  MoveL 8129 to (238.13, 41.99, 116.27) mm, rotated rx 180 ry 0 rz 180 deg; joints [-18.333, 8.057, 71.55, 61.436, 20.986, -59.754]
  Call Extruder(204.42198)
  MoveL 8130 to (238.31, 42.3, 116.27) mm, rotated rx 180 ry 0 rz 180 deg; joints [-18.36, 8.102, 71.5, 61.459, 21.011, -59.774]
  MoveL 8131 to (238.31, 42.3, 116.27) mm, rotated rx 180 ry 0 rz 180 deg; joints [-18.36, 8.102, 71.5, 61.459, 21.011, -59.774]
  Call Extruder(204.62931)
  MoveL 8132 to (238.49, 42.6, 116.27) mm, rotated rx 180 ry 0 rz 180 deg; joints [-18.386, 8.146, 71.449, 61.482, 21.037, -59.794]
  MoveL 8133 to (238.49, 42.6, 116.27) mm, rotated rx 180 ry 0 rz 180 deg; joints [-18.386, 8.146, 71.449, 61.482, 21.037, -59.794]
  Call Extruder(204.83587)
  MoveL 8134 to (238.66, 42.91, 116.27) mm, rotated rx 180 ry 0 rz 180 deg; joints [-18.412, 8.19, 71.399, 61.505, 21.062, -59.813]
  MoveL 8135 to (238.66, 42.91, 116.27) mm, rotated rx 180 ry 0 rz 180 deg; joints [-18.412, 8.19, 71.399, 61.505, 21.062, -59.813]
  Call Extruder(205.04165)
  MoveL 8136 to (238.84, 43.21, 116.27) mm, rotated rx 180 ry 0 rz -180 deg; joints [-18.438, 8.235, 71.349, 61.528, 21.088, -59.833]
  MoveL 8137 to (238.84, 43.21, 116.27) mm, rotated rx 180 ry 0 rz -180 deg; joints [-18.438, 8.235, 71.349, 61.528, 21.088, -59.833]
  Call Extruder(205.19996)
  MoveL 8138 to (238.94, 43.46, 116.27) mm, rotated rx 180 ry 0 rz 180 deg; joints [-18.461, 8.265, 71.314, 61.55, 21.11, -59.852]
  MoveL 8139 to (238.94, 43.46, 116.27) mm, rotated rx 180 ry 0 rz 180 deg; joints [-18.461, 8.265, 71.314, 61.55, 21.11, -59.852]
  Call Extruder(205.35767)
  MoveL 8140 to (239.05, 43.71, 116.27) mm, rotated rx 180 ry 0 rz 180 deg; joints [-18.484, 8.296, 71.279, 61.573, 21.131, -59.872]
  MoveL 8141 to (239.05, 43.71, 116.27) mm, rotated rx 180 ry 0 rz 180 deg; joints [-18.484, 8.296, 71.279, 61.573, 21.131, -59.872]
  Call Extruder(205.52776)
  MoveL 8142 to (239.16, 43.98, 116.27) mm, rotated rx 180 ry 0 rz 180 deg; joints [-18.509, 8.328, 71.242, 61.597, 21.155, -59.893]
  MoveL 8143 to (239.16, 43.98, 116.27) mm, rotated rx 180 ry 0 rz 180 deg; joints [-18.509, 8.328, 71.242, 61.597, 21.155, -59.893]
  Call Extruder(205.71010)
  MoveL 8144 to (239.29, 44.27, 116.27) mm, rotated rx 180 ry 0 rz -180 deg; joints [-18.535, 8.363, 71.202, 61.623, 21.18, -59.916]
  MoveL 8145 to (239.29, 44.27, 116.27) mm, rotated rx 180 ry 0 rz -180 deg; joints [-18.535, 8.363, 71.202, 61.623, 21.18, -59.916]
  Call Extruder(205.89168)
  MoveL 8146 to (239.41, 44.56, 116.27) mm, rotated rx 180 ry 0 rz 180 deg; joints [-18.562, 8.399, 71.162, 61.649, 21.206, -59.938]
  MoveL 8147 to (239.41, 44.56, 116.27) mm, rotated rx 180 ry 0 rz 180 deg; joints [-18.562, 8.399, 71.162, 61.649, 21.206, -59.938]
  Call Extruder(206.00513)
  MoveL 8148 to (239.47, 44.75, 116.27) mm, rotated rx -180 ry 0 rz 180 deg; joints [-18.58, 8.418, 71.139, 61.667, 21.223, -59.954]
  MoveL 8149 to (239.47, 44.75, 116.27) mm, rotated rx -180 ry 0 rz 180 deg; joints [-18.58, 8.418, 71.139, 61.667, 21.223, -59.954]
  Call Extruder(206.11815)
  MoveL 8150 to (239.53, 44.94, 116.27) mm, rotated rx 180 ry 0 rz 180 deg; joints [-18.598, 8.438, 71.116, 61.686, 21.239, -59.971]
  MoveL 8151 to (239.53, 44.94, 116.27) mm, rotated rx 180 ry 0 rz 180 deg; joints [-18.598, 8.438, 71.116, 61.686, 21.239, -59.971]
  Call Extruder(206.23072)
  MoveL 8152 to (239.59, 45.13, 116.27) mm, rotated rx 180 ry 0 rz -180 deg; joints [-18.616, 8.459, 71.093, 61.704, 21.256, -59.987]
  MoveL 8153 to (239.59, 45.13, 116.27) mm, rotated rx 180 ry 0 rz -180 deg; joints [-18.616, 8.459, 71.093, 61.704, 21.256, -59.987]
  Call Extruder(206.34284)
  MoveL 8154 to (239.65, 45.32, 116.27) mm, rotated rx -180 ry 0 rz 180 deg; joints [-18.634, 8.479, 71.071, 61.722, 21.273, -60.003]
  MoveL 8155 to (239.65, 45.32, 116.27) mm, rotated rx -180 ry 0 rz 180 deg; joints [-18.634, 8.479, 71.071, 61.722, 21.273, -60.003]
  Call Extruder(206.45452)
  MoveL 8156 to (239.71, 45.51, 116.27) mm, rotated rx -180 ry 0 rz 180 deg; joints [-18.651, 8.499, 71.048, 61.74, 21.29, -60.019]
  MoveL 8157 to (239.71, 45.51, 116.27) mm, rotated rx -180 ry 0 rz 180 deg; joints [-18.651, 8.499, 71.048, 61.74, 21.29, -60.019]
  Call Extruder(206.58559)
  MoveL 8158 to (239.78, 45.73, 116.27) mm, rotated rx 180 ry 0 rz 180 deg; joints [-18.673, 8.522, 71.022, 61.762, 21.31, -60.038]
  MoveL 8159 to (239.78, 45.73, 116.27) mm, rotated rx 180 ry 0 rz 180 deg; joints [-18.673, 8.522, 71.022, 61.762, 21.31, -60.038]
  Call Extruder(206.71610)
  MoveL 8160 to (239.85, 45.95, 116.27) mm, rotated rx 180 ry 0 rz -180 deg; joints [-18.694, 8.545, 70.995, 61.784, 21.33, -60.058]
  MoveL 8161 to (239.85, 45.95, 116.27) mm, rotated rx 180 ry 0 rz -180 deg; joints [-18.694, 8.545, 70.995, 61.784, 21.33, -60.058]
  Call Extruder(206.84604)
  MoveL 8162 to (239.92, 46.18, 116.27) mm, rotated rx 180 ry 0 rz -180 deg; joints [-18.715, 8.568, 70.969, 61.806, 21.35, -60.077]
  MoveL 8163 to (239.92, 46.18, 116.27) mm, rotated rx 180 ry 0 rz -180 deg; joints [-18.715, 8.568, 70.969, 61.806, 21.35, -60.077]
  Call Extruder(206.97542)
  MoveL 8164 to (239.98, 46.4, 116.27) mm, rotated rx -180 ry 0 rz -180 deg; joints [-18.737, 8.591, 70.943, 61.828, 21.37, -60.096]
  MoveL 8165 to (239.98, 46.4, 116.27) mm, rotated rx -180 ry 0 rz -180 deg; joints [-18.737, 8.591, 70.943, 61.828, 21.37, -60.096]
  Call Extruder(207.09738)
  MoveL 8166 to (240.04, 46.61, 116.27) mm, rotated rx -180 ry 0 rz 180 deg; joints [-18.757, 8.611, 70.919, 61.849, 21.389, -60.115]
  MoveL 8167 to (240.04, 46.61, 116.27) mm, rotated rx -180 ry 0 rz 180 deg; joints [-18.757, 8.611, 70.919, 61.849, 21.389, -60.115]
  Call Extruder(207.21220)
  MoveL 8168 to (240.08, 46.82, 116.27) mm, rotated rx 180 ry 0 rz 180 deg; joints [-18.777, 8.63, 70.898, 61.871, 21.408, -60.135]
  MoveL 8169 to (240.08, 46.82, 116.27) mm, rotated rx 180 ry 0 rz 180 deg; joints [-18.777, 8.63, 70.898, 61.871, 21.408, -60.135]
  Call Extruder(207.32658)
  MoveL 8170 to (240.13, 47.02, 116.27) mm, rotated rx -180 ry 0 rz 180 deg; joints [-18.797, 8.648, 70.877, 61.892, 21.426, -60.154]
  MoveL 8171 to (240.13, 47.02, 116.27) mm, rotated rx -180 ry 0 rz 180 deg; joints [-18.797, 8.648, 70.877, 61.892, 21.426, -60.154]
  Call Extruder(207.44050)
  MoveL 8172 to (240.17, 47.23, 116.27) mm, rotated rx 180 ry 0 rz 180 deg; joints [-18.817, 8.666, 70.856, 61.913, 21.445, -60.173]
  MoveL 8173 to (240.17, 47.23, 116.27) mm, rotated rx 180 ry 0 rz 180 deg; joints [-18.817, 8.666, 70.856, 61.913, 21.445, -60.173]
  Call Extruder(207.55397)
  MoveL 8174 to (240.22, 47.43, 116.27) mm, rotated rx 180 ry 0 rz 180 deg; joints [-18.837, 8.685, 70.835, 61.935, 21.464, -60.192]
  MoveL 8175 to (240.22, 47.43, 116.27) mm, rotated rx 180 ry 0 rz 180 deg; joints [-18.837, 8.685, 70.835, 61.935, 21.464, -60.192]
  Call Extruder(207.69125)
  MoveL 8176 to (240.27, 47.68, 116.27) mm, rotated rx 180 ry 0 rz -180 deg; joints [-18.862, 8.706, 70.81, 61.961, 21.486, -60.215]
  MoveL 8177 to (240.27, 47.68, 116.27) mm, rotated rx 180 ry 0 rz -180 deg; joints [-18.862, 8.706, 70.81, 61.961, 21.486, -60.215]
  Call Extruder(207.82792)
  MoveL 8178 to (240.32, 47.93, 116.27) mm, rotated rx 180 ry 0 rz 180 deg; joints [-18.887, 8.728, 70.786, 61.987, 21.509, -60.239]
  MoveL 8179 to (240.32, 47.93, 116.27) mm, rotated rx 180 ry 0 rz 180 deg; joints [-18.887, 8.728, 70.786, 61.987, 21.509, -60.239]
  Call Extruder(207.96399)
  MoveL 8180 to (240.37, 48.18, 116.27) mm, rotated rx 180 ry 0 rz 180 deg; joints [-18.911, 8.75, 70.761, 62.014, 21.532, -60.262]
  MoveL 8181 to (240.37, 48.18, 116.27) mm, rotated rx 180 ry 0 rz 180 deg; joints [-18.911, 8.75, 70.761, 62.014, 21.532, -60.262]
  Call Extruder(208.09944)
  MoveL 8182 to (240.42, 48.43, 116.27) mm, rotated rx 180 ry 0 rz 180 deg; joints [-18.936, 8.771, 70.736, 62.04, 21.555, -60.285]
  MoveL 8183 to (240.42, 48.43, 116.27) mm, rotated rx 180 ry 0 rz 180 deg; joints [-18.936, 8.771, 70.736, 62.04, 21.555, -60.285]
  Call Extruder(208.23428)
  MoveL 8184 to (240.47, 48.68, 116.27) mm, rotated rx 180 ry 0 rz -180 deg; joints [-18.96, 8.793, 70.711, 62.066, 21.578, -60.308]
  MoveL 8185 to (240.47, 48.68, 116.27) mm, rotated rx 180 ry 0 rz -180 deg; joints [-18.96, 8.793, 70.711, 62.066, 21.578, -60.308]
  Call Extruder(208.36851)
  MoveL 8186 to (240.52, 48.92, 116.27) mm, rotated rx 180 ry 0 rz 180 deg; joints [-18.985, 8.815, 70.686, 62.092, 21.6, -60.331]
  MoveL 8187 to (240.52, 48.92, 116.27) mm, rotated rx 180 ry 0 rz 180 deg; joints [-18.985, 8.815, 70.686, 62.092, 21.6, -60.331]
  Call Extruder(208.50213)
  MoveL 8188 to (240.57, 49.17, 116.27) mm, rotated rx 180 ry 0 rz 180 deg; joints [-19.009, 8.837, 70.661, 62.117, 21.623, -60.354]
  MoveL 8189 to (240.57, 49.17, 116.27) mm, rotated rx 180 ry 0 rz 180 deg; joints [-19.009, 8.837, 70.661, 62.117, 21.623, -60.354]
  Call Extruder(208.66424)
  MoveL 8190 to (240.61, 49.48, 116.27) mm, rotated rx -180 ry 0 rz 180 deg; joints [-19.04, 8.861, 70.633, 62.15, 21.651, -60.384]
  MoveL 8191 to (240.61, 49.48, 116.27) mm, rotated rx -180 ry 0 rz 180 deg; joints [-19.04, 8.861, 70.633, 62.15, 21.651, -60.384]
  Call Extruder(208.82562)
  MoveL 8192 to (240.66, 49.79, 116.27) mm, rotated rx 180 ry 0 rz 180 deg; joints [-19.07, 8.886, 70.604, 62.183, 21.68, -60.413]
  MoveL 8193 to (240.66, 49.79, 116.27) mm, rotated rx 180 ry 0 rz 180 deg; joints [-19.07, 8.886, 70.604, 62.183, 21.68, -60.413]
  Call Extruder(208.98628)
  MoveL 8194 to (240.71, 50.09, 116.27) mm, rotated rx 180 ry 0 rz 180 deg; joints [-19.101, 8.911, 70.576, 62.215, 21.708, -60.442]
  MoveL 8195 to (240.71, 50.09, 116.27) mm, rotated rx 180 ry 0 rz 180 deg; joints [-19.101, 8.911, 70.576, 62.215, 21.708, -60.442]
  Call Extruder(209.14620)
  MoveL 8196 to (240.76, 50.4, 116.27) mm, rotated rx 180 ry 0 rz 180 deg; joints [-19.131, 8.936, 70.547, 62.248, 21.736, -60.471]
  MoveL 8197 to (240.76, 50.4, 116.27) mm, rotated rx 180 ry 0 rz 180 deg; joints [-19.131, 8.936, 70.547, 62.248, 21.736, -60.471]
  Call Extruder(209.30540)
  MoveL 8198 to (240.81, 50.7, 116.27) mm, rotated rx 180 ry 0 rz -180 deg; joints [-19.162, 8.961, 70.519, 62.28, 21.764, -60.499]
  MoveL 8199 to (240.81, 50.7, 116.27) mm, rotated rx 180 ry 0 rz -180 deg; joints [-19.162, 8.961, 70.519, 62.28, 21.764, -60.499]
  Call Extruder(209.46387)
  MoveL 8200 to (240.86, 51.01, 116.27) mm, rotated rx 180 ry 0 rz 180 deg; joints [-19.192, 8.986, 70.49, 62.312, 21.793, -60.528]
  MoveL 8201 to (240.86, 51.01, 116.27) mm, rotated rx 180 ry 0 rz 180 deg; joints [-19.192, 8.986, 70.49, 62.312, 21.793, -60.528]
  Call Extruder(209.66274)
  MoveL 8202 to (240.9, 51.4, 116.27) mm, rotated rx 180 ry 0 rz 180 deg; joints [-19.231, 9.015, 70.457, 62.354, 21.829, -60.566]
  MoveL 8203 to (240.9, 51.4, 116.27) mm, rotated rx 180 ry 0 rz 180 deg; joints [-19.231, 9.015, 70.457, 62.354, 21.829, -60.566]
  Call Extruder(209.86075)
  MoveL 8204 to (240.95, 51.78, 116.27) mm, rotated rx 180 ry 0 rz 180 deg; joints [-19.27, 9.044, 70.423, 62.396, 21.865, -60.603]
  MoveL 8205 to (240.95, 51.78, 116.27) mm, rotated rx 180 ry 0 rz 180 deg; joints [-19.27, 9.044, 70.423, 62.396, 21.865, -60.603]
  Call Extruder(210.05789)
  MoveL 8206 to (240.99, 52.17, 116.27) mm, rotated rx 180 ry 0 rz -180 deg; joints [-19.309, 9.073, 70.389, 62.438, 21.901, -60.64]
  MoveL 8207 to (240.99, 52.17, 116.27) mm, rotated rx 180 ry 0 rz -180 deg; joints [-19.309, 9.073, 70.389, 62.438, 21.901, -60.64]
  Call Extruder(210.25416)
  MoveL 8208 to (241.04, 52.56, 116.27) mm, rotated rx 180 ry 0 rz 180 deg; joints [-19.348, 9.102, 70.356, 62.48, 21.937, -60.678]
  MoveL 8209 to (241.04, 52.56, 116.27) mm, rotated rx 180 ry 0 rz 180 deg; joints [-19.348, 9.102, 70.356, 62.48, 21.937, -60.678]
  Call Extruder(210.49987)
  MoveL 8210 to (241.09, 53.05, 116.27) mm, rotated rx 180 ry 0 rz 180 deg; joints [-19.398, 9.137, 70.315, 62.533, 21.983, -60.725]
  MoveL 8211 to (241.09, 53.05, 116.27) mm, rotated rx 180 ry 0 rz 180 deg; joints [-19.398, 9.137, 70.315, 62.533, 21.983, -60.725]
  Call Extruder(210.79465)
  MoveL 8212 to (241.13, 53.64, 116.27) mm, rotated rx 180 ry 0 rz 180 deg; joints [-19.458, 9.178, 70.268, 62.598, 22.038, -60.783]
  MoveL 8213 to (241.13, 53.64, 116.27) mm, rotated rx 180 ry 0 rz 180 deg; joints [-19.458, 9.178, 70.268, 62.598, 22.038, -60.783]
  Call Extruder(211.08809)
  MoveL 8214 to (241.18, 54.23, 116.27) mm, rotated rx 180 ry 0 rz 180 deg; joints [-19.518, 9.219, 70.221, 62.662, 22.093, -60.84]
  MoveL 8215 to (241.18, 54.23, 116.27) mm, rotated rx 180 ry 0 rz 180 deg; joints [-19.518, 9.219, 70.221, 62.662, 22.093, -60.84]
  Call Extruder(211.52144)
  MoveL 8216 to (241.22, 55.1, 116.27) mm, rotated rx 180 ry 0 rz 180 deg; joints [-19.608, 9.277, 70.154, 62.759, 22.176, -60.927]
  MoveL 8217 to (241.22, 55.1, 116.27) mm, rotated rx 180 ry 0 rz 180 deg; joints [-19.608, 9.277, 70.154, 62.759, 22.176, -60.927]
  Call Extruder(212.09360)
  MoveL 8218 to (241.27, 56.26, 116.27) mm, rotated rx 180 ry 0 rz 180 deg; joints [-19.728, 9.351, 70.069, 62.888, 22.286, -61.043]
  MoveL 8219 to (241.27, 56.26, 116.27) mm, rotated rx 180 ry 0 rz 180 deg; joints [-19.728, 9.351, 70.069, 62.888, 22.286, -61.043]
  Call Extruder(212.52130)
  MoveL 8220 to (241.29, 57.14, 116.27) mm, rotated rx 180 ry 0 rz 180 deg; joints [-19.819, 9.405, 70.007, 62.985, 22.369, -61.13]
  Call Extruder(254.51494)
  MoveL 8221 to (241.29, 142.86, 116.27) mm, rotated rx 180 ry 0 rz 180 deg; joints [-28.232, 15.645, 62.466, 69.008, 30.442, -66.009]
  MoveL 8222 to (241.29, 142.86, 116.27) mm, rotated rx 180 ry 0 rz 180 deg; joints [-28.232, 15.645, 62.466, 69.008, 30.442, -66.009]
  Call Extruder(255.23038)
  MoveL 8223 to (241.25, 144.32, 116.27) mm, rotated rx 180 ry 0 rz 180 deg; joints [-28.367, 15.768, 62.311, 69.066, 30.577, -66.043]
  MoveL 8224 to (241.25, 144.32, 116.27) mm, rotated rx 180 ry 0 rz 180 deg; joints [-28.367, 15.768, 62.311, 69.066, 30.577, -66.043]
  Call Extruder(255.80512)
  MoveL 8225 to (241.2, 145.48, 116.27) mm, rotated rx 180 ry 0 rz 180 deg; joints [-28.475, 15.864, 62.19, 69.112, 30.685, -66.071]
  MoveL 8226 to (241.2, 145.48, 116.27) mm, rotated rx 180 ry 0 rz 180 deg; joints [-28.475, 15.864, 62.19, 69.112, 30.685, -66.071]
  Call Extruder(256.09856)
  MoveL 8227 to (241.15, 146.07, 116.27) mm, rotated rx 180 ry 0 rz 180 deg; joints [-28.531, 15.909, 62.133, 69.138, 30.741, -66.087]
  MoveL 8228 to (241.15, 146.07, 116.27) mm, rotated rx 180 ry 0 rz 180 deg; joints [-28.531, 15.909, 62.133, 69.138, 30.741, -66.087]
  Call Extruder(256.39333)
  MoveL 8229 to (241.11, 146.66, 116.27) mm, rotated rx 180 ry 0 rz 180 deg; joints [-28.587, 15.954, 62.076, 69.163, 30.796, -66.103]
  MoveL 8230 to (241.11, 146.66, 116.27) mm, rotated rx 180 ry 0 rz 180 deg; joints [-28.587, 15.954, 62.076, 69.163, 30.796, -66.103]
  Call Extruder(256.68944)
  MoveL 8231 to (241.06, 147.25, 116.27) mm, rotated rx 180 ry 0 rz 180 deg; joints [-28.643, 15.999, 62.018, 69.189, 30.852, -66.119]
  MoveL 8232 to (241.06, 147.25, 116.27) mm, rotated rx 180 ry 0 rz 180 deg; joints [-28.643, 15.999, 62.018, 69.189, 30.852, -66.119]
  Call Extruder(256.88571)
  MoveL 8233 to (241.02, 147.63, 116.27) mm, rotated rx -180 ry 0 rz 180 deg; joints [-28.681, 16.027, 61.984, 69.207, 30.888, -66.131]
  MoveL 8234 to (241.02, 147.63, 116.27) mm, rotated rx -180 ry 0 rz 180 deg; joints [-28.681, 16.027, 61.984, 69.207, 30.888, -66.131]
  Call Extruder(257.08285)
  MoveL 8235 to (240.97, 148.02, 116.27) mm, rotated rx -180 ry 0 rz 180 deg; joints [-28.718, 16.054, 61.949, 69.225, 30.925, -66.143]
  MoveL 8236 to (240.97, 148.02, 116.27) mm, rotated rx -180 ry 0 rz 180 deg; joints [-28.718, 16.054, 61.949, 69.225, 30.925, -66.143]
  Call Extruder(257.28085)
  MoveL 8237 to (240.92, 148.41, 116.27) mm, rotated rx -180 ry 0 rz 180 deg; joints [-28.756, 16.082, 61.914, 69.243, 30.962, -66.155]
  MoveL 8238 to (240.92, 148.41, 116.27) mm, rotated rx -180 ry 0 rz 180 deg; joints [-28.756, 16.082, 61.914, 69.243, 30.962, -66.155]
  Call Extruder(257.47973)
  MoveL 8239 to (240.88, 148.8, 116.27) mm, rotated rx 180 ry 0 rz 180 deg; joints [-28.793, 16.109, 61.879, 69.261, 30.999, -66.167]
  MoveL 8240 to (240.88, 148.8, 116.27) mm, rotated rx 180 ry 0 rz 180 deg; joints [-28.793, 16.109, 61.879, 69.261, 30.999, -66.167]
  Call Extruder(257.65881)
  MoveL 8241 to (240.83, 149.14, 116.27) mm, rotated rx -180 ry 0 rz 180 deg; joints [-28.827, 16.133, 61.849, 69.277, 31.032, -66.178]
  MoveL 8242 to (240.83, 149.14, 116.27) mm, rotated rx -180 ry 0 rz 180 deg; joints [-28.827, 16.133, 61.849, 69.277, 31.032, -66.178]
  Call Extruder(257.81801)
  MoveL 8243 to (240.78, 149.45, 116.27) mm, rotated rx 180 ry 0 rz 180 deg; joints [-28.857, 16.153, 61.824, 69.293, 31.062, -66.189]
  MoveL 8244 to (240.78, 149.45, 116.27) mm, rotated rx 180 ry 0 rz 180 deg; joints [-28.857, 16.153, 61.824, 69.293, 31.062, -66.189]
  Call Extruder(257.97794)
  MoveL 8245 to (240.74, 149.76, 116.27) mm, rotated rx 180 ry 0 rz 180 deg; joints [-28.887, 16.173, 61.799, 69.308, 31.091, -66.199]
  MoveL 8246 to (240.74, 149.76, 116.27) mm, rotated rx 180 ry 0 rz 180 deg; joints [-28.887, 16.173, 61.799, 69.308, 31.091, -66.199]
  Call Extruder(258.13859)
  MoveL 8247 to (240.69, 150.06, 116.27) mm, rotated rx 180 ry 0 rz 180 deg; joints [-28.917, 16.192, 61.774, 69.323, 31.12, -66.21]
  MoveL 8248 to (240.69, 150.06, 116.27) mm, rotated rx 180 ry 0 rz 180 deg; joints [-28.917, 16.192, 61.774, 69.323, 31.12, -66.21]
  Call Extruder(258.29997)
  MoveL 8249 to (240.64, 150.37, 116.27) mm, rotated rx 180 ry 0 rz 180 deg; joints [-28.947, 16.212, 61.749, 69.338, 31.15, -66.22]
  MoveL 8250 to (240.64, 150.37, 116.27) mm, rotated rx 180 ry 0 rz 180 deg; joints [-28.947, 16.212, 61.749, 69.338, 31.15, -66.22]
  Call Extruder(258.46208)
  MoveL 8251 to (240.59, 150.67, 116.27) mm, rotated rx -180 ry 0 rz 180 deg; joints [-28.978, 16.232, 61.723, 69.353, 31.179, -66.23]
  MoveL 8252 to (240.59, 150.67, 116.27) mm, rotated rx -180 ry 0 rz 180 deg; joints [-28.978, 16.232, 61.723, 69.353, 31.179, -66.23]
  Call Extruder(258.61028)
  MoveL 8253 to (240.54, 150.95, 116.27) mm, rotated rx -180 ry 0 rz 180 deg; joints [-29.005, 16.249, 61.701, 69.368, 31.206, -66.24]
  MoveL 8254 to (240.54, 150.95, 116.27) mm, rotated rx -180 ry 0 rz 180 deg; joints [-29.005, 16.249, 61.701, 69.368, 31.206, -66.24]
  Call Extruder(258.74452)
  MoveL 8255 to (240.49, 151.2, 116.27) mm, rotated rx 180 ry 0 rz 180 deg; joints [-29.03, 16.264, 61.683, 69.381, 31.23, -66.25]
  MoveL 8256 to (240.49, 151.2, 116.27) mm, rotated rx 180 ry 0 rz 180 deg; joints [-29.03, 16.264, 61.683, 69.381, 31.23, -66.25]
  Call Extruder(258.87936)
  MoveL 8257 to (240.44, 151.45, 116.27) mm, rotated rx 180 ry 0 rz 180 deg; joints [-29.055, 16.279, 61.664, 69.394, 31.255, -66.259]
  MoveL 8258 to (240.44, 151.45, 116.27) mm, rotated rx 180 ry 0 rz 180 deg; joints [-29.055, 16.279, 61.664, 69.394, 31.255, -66.259]
  Call Extruder(259.01481)
  MoveL 8259 to (240.39, 151.7, 116.27) mm, rotated rx -180 ry 0 rz 180 deg; joints [-29.08, 16.293, 61.646, 69.407, 31.279, -66.268]
  MoveL 8260 to (240.39, 151.7, 116.27) mm, rotated rx -180 ry 0 rz 180 deg; joints [-29.08, 16.293, 61.646, 69.407, 31.279, -66.268]
  Call Extruder(259.15087)
  MoveL 8261 to (240.34, 151.95, 116.27) mm, rotated rx 180 ry 0 rz 180 deg; joints [-29.105, 16.308, 61.627, 69.421, 31.303, -66.278]
  MoveL 8262 to (240.34, 151.95, 116.27) mm, rotated rx 180 ry 0 rz 180 deg; joints [-29.105, 16.308, 61.627, 69.421, 31.303, -66.278]
  Call Extruder(259.28754)
  MoveL 8263 to (240.29, 152.2, 116.27) mm, rotated rx 180 ry 0 rz 180 deg; joints [-29.13, 16.323, 61.608, 69.434, 31.327, -66.287]
  MoveL 8264 to (240.29, 152.2, 116.27) mm, rotated rx 180 ry 0 rz 180 deg; joints [-29.13, 16.323, 61.608, 69.434, 31.327, -66.287]
  Call Extruder(259.42483)
  MoveL 8265 to (240.24, 152.44, 116.27) mm, rotated rx 180 ry 0 rz 180 deg; joints [-29.155, 16.338, 61.589, 69.447, 31.352, -66.296]
  MoveL 8266 to (240.24, 152.44, 116.27) mm, rotated rx 180 ry 0 rz 180 deg; joints [-29.155, 16.338, 61.589, 69.447, 31.352, -66.296]
  Call Extruder(259.55049)
  MoveL 8267 to (240.2, 152.67, 116.27) mm, rotated rx -180 ry 0 rz 180 deg; joints [-29.178, 16.351, 61.573, 69.459, 31.374, -66.305]
  MoveL 8268 to (240.2, 152.67, 116.27) mm, rotated rx -180 ry 0 rz 180 deg; joints [-29.178, 16.351, 61.573, 69.459, 31.374, -66.305]
  Call Extruder(259.66441)
  MoveL 8269 to (240.15, 152.88, 116.27) mm, rotated rx 180 ry 0 rz -180 deg; joints [-29.198, 16.362, 61.558, 69.47, 31.394, -66.313]
  MoveL 8270 to (240.15, 152.88, 116.27) mm, rotated rx 180 ry 0 rz -180 deg; joints [-29.198, 16.362, 61.558, 69.47, 31.394, -66.313]
  Call Extruder(259.77879)
  MoveL 8271 to (240.11, 153.08, 116.27) mm, rotated rx 180 ry 0 rz 180 deg; joints [-29.219, 16.374, 61.543, 69.481, 31.414, -66.321]
  MoveL 8272 to (240.11, 153.08, 116.27) mm, rotated rx 180 ry 0 rz 180 deg; joints [-29.219, 16.374, 61.543, 69.481, 31.414, -66.321]
  Call Extruder(259.89362)
  MoveL 8273 to (240.06, 153.28, 116.27) mm, rotated rx 180 ry 0 rz 180 deg; joints [-29.24, 16.385, 61.529, 69.492, 31.434, -66.329]
  MoveL 8274 to (240.06, 153.28, 116.27) mm, rotated rx 180 ry 0 rz 180 deg; joints [-29.24, 16.385, 61.529, 69.492, 31.434, -66.329]
  Call Extruder(260.00890)
  MoveL 8275 to (240.02, 153.49, 116.27) mm, rotated rx -180 ry 0 rz 180 deg; joints [-29.26, 16.396, 61.514, 69.503, 31.454, -66.337]
  MoveL 8276 to (240.02, 153.49, 116.27) mm, rotated rx -180 ry 0 rz 180 deg; joints [-29.26, 16.396, 61.514, 69.503, 31.454, -66.337]
  Call Extruder(260.13828)
  MoveL 8277 to (239.95, 153.71, 116.27) mm, rotated rx -180 ry 0 rz 180 deg; joints [-29.284, 16.406, 61.502, 69.518, 31.476, -66.347]
  MoveL 8278 to (239.95, 153.71, 116.27) mm, rotated rx -180 ry 0 rz 180 deg; joints [-29.284, 16.406, 61.502, 69.518, 31.476, -66.347]
  Call Extruder(260.26822)
  MoveL 8279 to (239.88, 153.94, 116.27) mm, rotated rx -180 ry 0 rz 180 deg; joints [-29.307, 16.416, 61.49, 69.532, 31.499, -66.358]
  MoveL 8280 to (239.88, 153.94, 116.27) mm, rotated rx -180 ry 0 rz 180 deg; joints [-29.307, 16.416, 61.49, 69.532, 31.499, -66.358]
  Call Extruder(260.39873)
  MoveL 8281 to (239.82, 154.16, 116.27) mm, rotated rx 180 ry 0 rz 180 deg; joints [-29.331, 16.425, 61.478, 69.546, 31.521, -66.369]
  MoveL 8282 to (239.82, 154.16, 116.27) mm, rotated rx 180 ry 0 rz 180 deg; joints [-29.331, 16.425, 61.478, 69.546, 31.521, -66.369]
  Call Extruder(260.52980)
  MoveL 8283 to (239.75, 154.38, 116.27) mm, rotated rx -180 ry 0 rz 180 deg; joints [-29.354, 16.435, 61.466, 69.56, 31.544, -66.38]
  MoveL 8284 to (239.75, 154.38, 116.27) mm, rotated rx -180 ry 0 rz 180 deg; joints [-29.354, 16.435, 61.466, 69.56, 31.544, -66.38]
  Call Extruder(260.65144)
  MoveL 8285 to (239.68, 154.59, 116.27) mm, rotated rx 180 ry 0 rz 180 deg; joints [-29.376, 16.443, 61.455, 69.573, 31.565, -66.39]
  MoveL 8286 to (239.68, 154.59, 116.27) mm, rotated rx 180 ry 0 rz 180 deg; joints [-29.376, 16.443, 61.455, 69.573, 31.565, -66.39]
  Call Extruder(260.76357)
  MoveL 8287 to (239.62, 154.78, 116.27) mm, rotated rx 180 ry 0 rz 180 deg; joints [-29.396, 16.451, 61.445, 69.585, 31.584, -66.399]
  MoveL 8288 to (239.62, 154.78, 116.27) mm, rotated rx 180 ry 0 rz 180 deg; joints [-29.396, 16.451, 61.445, 69.585, 31.584, -66.399]
  Call Extruder(260.87613)
  MoveL 8289 to (239.56, 154.97, 116.27) mm, rotated rx 180 ry 0 rz 180 deg; joints [-29.416, 16.458, 61.436, 69.597, 31.603, -66.408]
  MoveL 8290 to (239.56, 154.97, 116.27) mm, rotated rx 180 ry 0 rz 180 deg; joints [-29.416, 16.458, 61.436, 69.597, 31.603, -66.408]
  Call Extruder(260.98915)
  MoveL 8291 to (239.5, 155.15, 116.27) mm, rotated rx 180 ry 0 rz 180 deg; joints [-29.436, 16.466, 61.426, 69.609, 31.622, -66.418]
  MoveL 8292 to (239.5, 155.15, 116.27) mm, rotated rx 180 ry 0 rz 180 deg; joints [-29.436, 16.466, 61.426, 69.609, 31.622, -66.418]
  Call Extruder(261.10260)
  MoveL 8293 to (239.44, 155.34, 116.27) mm, rotated rx 180 ry 0 rz 180 deg; joints [-29.456, 16.473, 61.417, 69.622, 31.641, -66.427]
  MoveL 8294 to (239.44, 155.34, 116.27) mm, rotated rx 180 ry 0 rz 180 deg; joints [-29.456, 16.473, 61.417, 69.622, 31.641, -66.427]
  Call Extruder(261.25025)
  MoveL 8295 to (239.35, 155.58, 116.27) mm, rotated rx 180 ry 0 rz -180 deg; joints [-29.483, 16.48, 61.408, 69.639, 31.666, -66.441]
  MoveL 8296 to (239.35, 155.58, 116.27) mm, rotated rx 180 ry 0 rz -180 deg; joints [-29.483, 16.48, 61.408, 69.639, 31.666, -66.441]
  Call Extruder(261.43258)
  MoveL 8297 to (239.22, 155.88, 116.27) mm, rotated rx 180 ry 0 rz 180 deg; joints [-29.515, 16.488, 61.398, 69.66, 31.696, -66.458]
  MoveL 8298 to (239.22, 155.88, 116.27) mm, rotated rx 180 ry 0 rz 180 deg; joints [-29.515, 16.488, 61.398, 69.66, 31.696, -66.458]
  Call Extruder(261.61568)
  MoveL 8299 to (239.11, 156.17, 116.27) mm, rotated rx 180 ry 0 rz 180 deg; joints [-29.547, 16.495, 61.389, 69.682, 31.726, -66.475]
  MoveL 8300 to (239.11, 156.17, 116.27) mm, rotated rx 180 ry 0 rz 180 deg; joints [-29.547, 16.495, 61.389, 69.682, 31.726, -66.475]
  Call Extruder(261.77338)
  MoveL 8301 to (239, 156.42, 116.27) mm, rotated rx 180 ry 0 rz 180 deg; joints [-29.575, 16.501, 61.382, 69.7, 31.752, -66.49]
  MoveL 8302 to (239, 156.42, 116.27) mm, rotated rx 180 ry 0 rz 180 deg; joints [-29.575, 16.501, 61.382, 69.7, 31.752, -66.49]
  Call Extruder(261.93170)
  MoveL 8303 to (238.89, 156.66, 116.27) mm, rotated rx -180 ry 0 rz 180 deg; joints [-29.603, 16.506, 61.374, 69.719, 31.778, -66.505]
  MoveL 8304 to (238.89, 156.66, 116.27) mm, rotated rx -180 ry 0 rz 180 deg; joints [-29.603, 16.506, 61.374, 69.719, 31.778, -66.505]
  Call Extruder(262.11373)
  MoveL 8305 to (238.75, 156.94, 116.27) mm, rotated rx 180 ry 0 rz 180 deg; joints [-29.635, 16.509, 61.371, 69.742, 31.808, -66.525]
  MoveL 8306 to (238.75, 156.94, 116.27) mm, rotated rx 180 ry 0 rz 180 deg; joints [-29.635, 16.509, 61.371, 69.742, 31.808, -66.525]
  Call Extruder(262.32029)
  MoveL 8307 to (238.57, 157.25, 116.27) mm, rotated rx -180 ry 0 rz 180 deg; joints [-29.671, 16.509, 61.372, 69.77, 31.841, -66.548]
  MoveL 8308 to (238.57, 157.25, 116.27) mm, rotated rx -180 ry 0 rz 180 deg; joints [-29.671, 16.509, 61.372, 69.77, 31.841, -66.548]
  Call Extruder(262.52763)
  MoveL 8309 to (238.4, 157.55, 116.27) mm, rotated rx 180 ry 0 rz 180 deg; joints [-29.707, 16.508, 61.372, 69.797, 31.874, -66.571]
  MoveL 8310 to (238.4, 157.55, 116.27) mm, rotated rx 180 ry 0 rz 180 deg; joints [-29.707, 16.508, 61.372, 69.797, 31.874, -66.571]
  Call Extruder(262.73575)
  MoveL 8311 to (238.22, 157.85, 116.27) mm, rotated rx 180 ry 0 rz 180 deg; joints [-29.743, 16.508, 61.372, 69.824, 31.907, -66.595]
  MoveL 8312 to (238.22, 157.85, 116.27) mm, rotated rx 180 ry 0 rz 180 deg; joints [-29.743, 16.508, 61.372, 69.824, 31.907, -66.595]
  Call Extruder(262.85347)
  MoveL 8313 to (238.12, 158.03, 116.27) mm, rotated rx 180 ry 0 rz 180 deg; joints [-29.764, 16.508, 61.373, 69.84, 31.926, -66.608]
  MoveL 8314 to (238.12, 158.03, 116.27) mm, rotated rx 180 ry 0 rz 180 deg; joints [-29.764, 16.508, 61.373, 69.84, 31.926, -66.608]
  Call Extruder(263.18629)
  MoveL 8315 to (237.79, 158.48, 116.27) mm, rotated rx 180 ry 0 rz 180 deg; joints [-29.821, 16.496, 61.387, 69.887, 31.977, -66.65]
  MoveL 8316 to (237.79, 158.48, 116.27) mm, rotated rx 180 ry 0 rz 180 deg; joints [-29.821, 16.496, 61.387, 69.887, 31.977, -66.65]
  Call Extruder(263.52029)
  MoveL 8317 to (237.47, 158.93, 116.27) mm, rotated rx 180 ry 0 rz -180 deg; joints [-29.878, 16.485, 61.402, 69.935, 32.029, -66.692]
  MoveL 8318 to (237.47, 158.93, 116.27) mm, rotated rx 180 ry 0 rz -180 deg; joints [-29.878, 16.485, 61.402, 69.935, 32.029, -66.692]
  Call Extruder(263.68786)
  MoveL 8319 to (237.3, 159.15, 116.27) mm, rotated rx -180 ry 0 rz -180 deg; joints [-29.907, 16.479, 61.409, 69.959, 32.055, -66.712]
  Call Extruder(264.51719)
  MoveL 8320 to (236.39, 160.19, 116.27) mm, rotated rx 180 ry 0 rz 180 deg; joints [-30.046, 16.428, 61.475, 70.083, 32.178, -66.825]
  Call Extruder(265.14825)
  MoveL 8321 to (235.6, 160.89, 116.27) mm, rotated rx 180 ry 0 rz -180 deg; joints [-30.149, 16.365, 61.554, 70.185, 32.267, -66.919]
  MoveL 8322 to (235.6, 160.89, 116.27) mm, rotated rx 180 ry 0 rz -180 deg; joints [-30.149, 16.365, 61.554, 70.185, 32.267, -66.919]
  Call Extruder(265.34587)
  MoveL 8323 to (235.35, 161.1, 116.27) mm, rotated rx -180 ry 0 rz 180 deg; joints [-30.182, 16.345, 61.58, 70.217, 32.295, -66.949]
  Call Extruder(265.67988)
  MoveL 8324 to (234.9, 161.43, 116.27) mm, rotated rx 180 ry 0 rz 180 deg; joints [-30.234, 16.302, 61.635, 70.272, 32.339, -67.002]
  MoveL 8325 to (234.9, 161.43, 116.27) mm, rotated rx 180 ry 0 rz 180 deg; joints [-30.234, 16.302, 61.635, 70.272, 32.339, -67.002]
  Call Extruder(266.01272)
  MoveL 8326 to (234.45, 161.76, 116.27) mm, rotated rx -180 ry 0 rz 180 deg; joints [-30.287, 16.26, 61.688, 70.328, 32.384, -67.055]
  MoveL 8327 to (234.45, 161.76, 116.27) mm, rotated rx -180 ry 0 rz 180 deg; joints [-30.287, 16.26, 61.688, 70.328, 32.384, -67.055]
  Call Extruder(266.19191)
  MoveL 8328 to (234.21, 161.93, 116.27) mm, rotated rx 180 ry 0 rz 180 deg; joints [-30.316, 16.236, 61.718, 70.358, 32.408, -67.083]
  MoveL 8329 to (234.21, 161.93, 116.27) mm, rotated rx 180 ry 0 rz 180 deg; joints [-30.316, 16.236, 61.718, 70.358, 32.408, -67.083]
  Call Extruder(266.40003)
  MoveL 8330 to (233.9, 162.11, 116.27) mm, rotated rx 180 ry 0 rz 180 deg; joints [-30.347, 16.204, 61.759, 70.394, 32.434, -67.118]
  MoveL 8331 to (233.9, 162.11, 116.27) mm, rotated rx 180 ry 0 rz 180 deg; joints [-30.347, 16.204, 61.759, 70.394, 32.434, -67.118]
  Call Extruder(266.60737)
  MoveL 8332 to (233.6, 162.29, 116.27) mm, rotated rx 180 ry 0 rz 180 deg; joints [-30.379, 16.171, 61.801, 70.43, 32.46, -67.153]
  MoveL 8333 to (233.6, 162.29, 116.27) mm, rotated rx 180 ry 0 rz 180 deg; joints [-30.379, 16.171, 61.801, 70.43, 32.46, -67.153]
  Call Extruder(266.81392)
  MoveL 8334 to (233.29, 162.46, 116.27) mm, rotated rx -180 ry 0 rz 180 deg; joints [-30.41, 16.138, 61.842, 70.466, 32.487, -67.188]
  MoveL 8335 to (233.29, 162.46, 116.27) mm, rotated rx -180 ry 0 rz 180 deg; joints [-30.41, 16.138, 61.842, 70.466, 32.487, -67.188]
  Call Extruder(267.01970)
  MoveL 8336 to (232.99, 162.64, 116.27) mm, rotated rx 180 ry 0 rz 180 deg; joints [-30.442, 16.106, 61.884, 70.501, 32.513, -67.222]
  MoveL 8337 to (232.99, 162.64, 116.27) mm, rotated rx 180 ry 0 rz 180 deg; joints [-30.442, 16.106, 61.884, 70.501, 32.513, -67.222]
  Call Extruder(267.17798)
  MoveL 8338 to (232.74, 162.74, 116.27) mm, rotated rx 180 ry 0 rz 180 deg; joints [-30.464, 16.076, 61.922, 70.53, 32.531, -67.25]
  MoveL 8339 to (232.74, 162.74, 116.27) mm, rotated rx 180 ry 0 rz 180 deg; joints [-30.464, 16.076, 61.922, 70.53, 32.531, -67.25]
  Call Extruder(267.33565)
  MoveL 8340 to (232.49, 162.85, 116.27) mm, rotated rx 180 ry 0 rz 180 deg; joints [-30.487, 16.045, 61.96, 70.558, 32.549, -67.278]
  MoveL 8341 to (232.49, 162.85, 116.27) mm, rotated rx 180 ry 0 rz 180 deg; joints [-30.487, 16.045, 61.96, 70.558, 32.549, -67.278]
  Call Extruder(267.50574)
  MoveL 8342 to (232.22, 162.97, 116.27) mm, rotated rx -180 ry 0 rz 180 deg; joints [-30.511, 16.012, 62.002, 70.588, 32.569, -67.308]
  MoveL 8343 to (232.22, 162.97, 116.27) mm, rotated rx -180 ry 0 rz 180 deg; joints [-30.511, 16.012, 62.002, 70.588, 32.569, -67.308]
  Call Extruder(267.68811)
  MoveL 8344 to (231.93, 163.09, 116.27) mm, rotated rx -180 ry 0 rz 180 deg; joints [-30.538, 15.977, 62.047, 70.621, 32.59, -67.341]
  MoveL 8345 to (231.93, 163.09, 116.27) mm, rotated rx -180 ry 0 rz 180 deg; joints [-30.538, 15.977, 62.047, 70.621, 32.59, -67.341]
  Call Extruder(267.86971)
  MoveL 8346 to (231.64, 163.21, 116.27) mm, rotated rx 180 ry 0 rz 180 deg; joints [-30.564, 15.941, 62.092, 70.654, 32.611, -67.373]
  MoveL 8347 to (231.64, 163.21, 116.27) mm, rotated rx 180 ry 0 rz 180 deg; joints [-30.564, 15.941, 62.092, 70.654, 32.611, -67.373]
  Call Extruder(267.98315)
  MoveL 8348 to (231.45, 163.27, 116.27) mm, rotated rx 180 ry 0 rz 180 deg; joints [-30.579, 15.916, 62.124, 70.674, 32.623, -67.394]
  MoveL 8349 to (231.45, 163.27, 116.27) mm, rotated rx 180 ry 0 rz 180 deg; joints [-30.579, 15.916, 62.124, 70.674, 32.623, -67.394]
  Call Extruder(268.09615)
  MoveL 8350 to (231.26, 163.33, 116.27) mm, rotated rx 180 ry 0 rz 180 deg; joints [-30.595, 15.892, 62.155, 70.695, 32.635, -67.414]
  MoveL 8351 to (231.26, 163.33, 116.27) mm, rotated rx 180 ry 0 rz 180 deg; joints [-30.595, 15.892, 62.155, 70.695, 32.635, -67.414]
  Call Extruder(268.20871)
  MoveL 8352 to (231.07, 163.39, 116.27) mm, rotated rx 180 ry 0 rz 180 deg; joints [-30.61, 15.867, 62.186, 70.715, 32.647, -67.435]
  MoveL 8353 to (231.07, 163.39, 116.27) mm, rotated rx 180 ry 0 rz 180 deg; joints [-30.61, 15.867, 62.186, 70.715, 32.647, -67.435]
  Call Extruder(268.32082)
  MoveL 8354 to (230.88, 163.45, 116.27) mm, rotated rx 180 ry 0 rz -180 deg; joints [-30.625, 15.843, 62.217, 70.736, 32.659, -67.456]
  MoveL 8355 to (230.88, 163.45, 116.27) mm, rotated rx 180 ry 0 rz -180 deg; joints [-30.625, 15.843, 62.217, 70.736, 32.659, -67.456]
  Call Extruder(268.43249)
  MoveL 8356 to (230.69, 163.51, 116.27) mm, rotated rx 180 ry 0 rz 180 deg; joints [-30.641, 15.818, 62.248, 70.756, 32.671, -67.476]
  MoveL 8357 to (230.69, 163.51, 116.27) mm, rotated rx 180 ry 0 rz 180 deg; joints [-30.641, 15.818, 62.248, 70.756, 32.671, -67.476]
  Call Extruder(268.56358)
  MoveL 8358 to (230.47, 163.58, 116.27) mm, rotated rx 180 ry 0 rz 180 deg; joints [-30.659, 15.789, 62.285, 70.781, 32.685, -67.5]
  MoveL 8359 to (230.47, 163.58, 116.27) mm, rotated rx 180 ry 0 rz 180 deg; joints [-30.659, 15.789, 62.285, 70.781, 32.685, -67.5]
  Call Extruder(268.69411)
  MoveL 8360 to (230.25, 163.65, 116.27) mm, rotated rx 180 ry 0 rz 180 deg; joints [-30.677, 15.759, 62.323, 70.805, 32.699, -67.525]
  MoveL 8361 to (230.25, 163.65, 116.27) mm, rotated rx 180 ry 0 rz 180 deg; joints [-30.677, 15.759, 62.323, 70.805, 32.699, -67.525]
  Call Extruder(268.82408)
  MoveL 8362 to (230.02, 163.72, 116.27) mm, rotated rx 180 ry 0 rz 180 deg; joints [-30.694, 15.73, 62.36, 70.829, 32.713, -67.549]
  MoveL 8363 to (230.02, 163.72, 116.27) mm, rotated rx 180 ry 0 rz 180 deg; joints [-30.694, 15.73, 62.36, 70.829, 32.713, -67.549]
  Call Extruder(268.95347)
  MoveL 8364 to (229.8, 163.78, 116.27) mm, rotated rx 180 ry 0 rz 180 deg; joints [-30.712, 15.7, 62.397, 70.853, 32.727, -67.573]
  MoveL 8365 to (229.8, 163.78, 116.27) mm, rotated rx 180 ry 0 rz 180 deg; joints [-30.712, 15.7, 62.397, 70.853, 32.727, -67.573]
  Call Extruder(269.07545)
  MoveL 8366 to (229.59, 163.84, 116.27) mm, rotated rx 180 ry 0 rz 180 deg; joints [-30.729, 15.671, 62.434, 70.875, 32.74, -67.596]
  MoveL 8367 to (229.59, 163.84, 116.27) mm, rotated rx 180 ry 0 rz 180 deg; joints [-30.729, 15.671, 62.434, 70.875, 32.74, -67.596]
  Call Extruder(269.19030)
  MoveL 8368 to (229.38, 163.88, 116.27) mm, rotated rx 180 ry 0 rz 180 deg; joints [-30.744, 15.642, 62.47, 70.897, 32.751, -67.618]
  MoveL 8369 to (229.38, 163.88, 116.27) mm, rotated rx 180 ry 0 rz 180 deg; joints [-30.744, 15.642, 62.47, 70.897, 32.751, -67.618]
  Call Extruder(269.30469)
  MoveL 8370 to (229.18, 163.93, 116.27) mm, rotated rx -180 ry 0 rz 180 deg; joints [-30.758, 15.614, 62.505, 70.918, 32.762, -67.639]
  MoveL 8371 to (229.18, 163.93, 116.27) mm, rotated rx -180 ry 0 rz 180 deg; joints [-30.758, 15.614, 62.505, 70.918, 32.762, -67.639]
  Call Extruder(269.41863)
  MoveL 8372 to (228.97, 163.97, 116.27) mm, rotated rx -180 ry 0 rz 180 deg; joints [-30.773, 15.585, 62.541, 70.94, 32.774, -67.661]
  MoveL 8373 to (228.97, 163.97, 116.27) mm, rotated rx -180 ry 0 rz 180 deg; joints [-30.773, 15.585, 62.541, 70.94, 32.774, -67.661]
  Call Extruder(269.53212)
  MoveL 8374 to (228.77, 164.02, 116.27) mm, rotated rx 180 ry 0 rz 180 deg; joints [-30.788, 15.557, 62.577, 70.961, 32.785, -67.683]
  MoveL 8375 to (228.77, 164.02, 116.27) mm, rotated rx 180 ry 0 rz 180 deg; joints [-30.788, 15.557, 62.577, 70.961, 32.785, -67.683]
  Call Extruder(269.66941)
  MoveL 8376 to (228.52, 164.07, 116.27) mm, rotated rx 180 ry 0 rz 180 deg; joints [-30.806, 15.522, 62.621, 70.987, 32.798, -67.709]
  MoveL 8377 to (228.52, 164.07, 116.27) mm, rotated rx 180 ry 0 rz 180 deg; joints [-30.806, 15.522, 62.621, 70.987, 32.798, -67.709]
  Call Extruder(269.80608)
  MoveL 8378 to (228.27, 164.12, 116.27) mm, rotated rx -180 ry 0 rz 180 deg; joints [-30.823, 15.487, 62.666, 71.012, 32.812, -67.735]
  MoveL 8379 to (228.27, 164.12, 116.27) mm, rotated rx -180 ry 0 rz 180 deg; joints [-30.823, 15.487, 62.666, 71.012, 32.812, -67.735]
  Call Extruder(269.94214)
  MoveL 8380 to (228.02, 164.17, 116.27) mm, rotated rx 180 ry 0 rz 180 deg; joints [-30.841, 15.452, 62.71, 71.038, 32.825, -67.762]
  MoveL 8381 to (228.02, 164.17, 116.27) mm, rotated rx 180 ry 0 rz 180 deg; joints [-30.841, 15.452, 62.71, 71.038, 32.825, -67.762]
  Call Extruder(270.07759)
  MoveL 8382 to (227.77, 164.22, 116.27) mm, rotated rx 180 ry 0 rz 180 deg; joints [-30.859, 15.417, 62.754, 71.063, 32.839, -67.788]
  MoveL 8383 to (227.77, 164.22, 116.27) mm, rotated rx 180 ry 0 rz 180 deg; joints [-30.859, 15.417, 62.754, 71.063, 32.839, -67.788]
  Call Extruder(270.21244)
  MoveL 8384 to (227.52, 164.27, 116.27) mm, rotated rx -180 ry 0 rz 180 deg; joints [-30.877, 15.382, 62.798, 71.089, 32.852, -67.814]
  MoveL 8385 to (227.52, 164.27, 116.27) mm, rotated rx -180 ry 0 rz 180 deg; joints [-30.877, 15.382, 62.798, 71.089, 32.852, -67.814]
  Call Extruder(270.34667)
  MoveL 8386 to (227.27, 164.32, 116.27) mm, rotated rx 180 ry 0 rz 180 deg; joints [-30.895, 15.347, 62.842, 71.114, 32.866, -67.84]
  MoveL 8387 to (227.27, 164.32, 116.27) mm, rotated rx 180 ry 0 rz 180 deg; joints [-30.895, 15.347, 62.842, 71.114, 32.866, -67.84]
  Call Extruder(270.48029)
  MoveL 8388 to (227.02, 164.37, 116.27) mm, rotated rx 180 ry 0 rz 180 deg; joints [-30.912, 15.311, 62.886, 71.14, 32.879, -67.866]
  MoveL 8389 to (227.02, 164.37, 116.27) mm, rotated rx 180 ry 0 rz 180 deg; joints [-30.912, 15.311, 62.886, 71.14, 32.879, -67.866]
  Call Extruder(270.64240)
  MoveL 8390 to (226.72, 164.41, 116.27) mm, rotated rx 180 ry 0 rz 180 deg; joints [-30.933, 15.268, 62.941, 71.171, 32.895, -67.897]
  MoveL 8391 to (226.72, 164.41, 116.27) mm, rotated rx 180 ry 0 rz 180 deg; joints [-30.933, 15.268, 62.941, 71.171, 32.895, -67.897]
  Call Extruder(270.80377)
  MoveL 8392 to (226.41, 164.46, 116.27) mm, rotated rx 180 ry 0 rz -180 deg; joints [-30.954, 15.223, 62.996, 71.201, 32.911, -67.929]
  MoveL 8393 to (226.41, 164.46, 116.27) mm, rotated rx 180 ry 0 rz -180 deg; joints [-30.954, 15.223, 62.996, 71.201, 32.911, -67.929]
  Call Extruder(270.96442)
  MoveL 8394 to (226.11, 164.51, 116.27) mm, rotated rx -180 ry 0 rz -180 deg; joints [-30.975, 15.179, 63.051, 71.232, 32.926, -67.96]
  MoveL 8395 to (226.11, 164.51, 116.27) mm, rotated rx -180 ry 0 rz -180 deg; joints [-30.975, 15.179, 63.051, 71.232, 32.926, -67.96]
  Call Extruder(271.12435)
  MoveL 8396 to (225.8, 164.56, 116.27) mm, rotated rx 180 ry 0 rz -180 deg; joints [-30.995, 15.136, 63.106, 71.262, 32.942, -67.992]
  MoveL 8397 to (225.8, 164.56, 116.27) mm, rotated rx 180 ry 0 rz -180 deg; joints [-30.995, 15.136, 63.106, 71.262, 32.942, -67.992]
  Call Extruder(271.28354)
  MoveL 8398 to (225.5, 164.61, 116.27) mm, rotated rx -180 ry 0 rz 180 deg; joints [-31.016, 15.092, 63.161, 71.293, 32.958, -68.023]
  MoveL 8399 to (225.5, 164.61, 116.27) mm, rotated rx -180 ry 0 rz 180 deg; joints [-31.016, 15.092, 63.161, 71.293, 32.958, -68.023]
  Call Extruder(271.44201)
  MoveL 8400 to (225.19, 164.66, 116.27) mm, rotated rx 180 ry 0 rz -180 deg; joints [-31.037, 15.048, 63.216, 71.323, 32.973, -68.054]
  MoveL 8401 to (225.19, 164.66, 116.27) mm, rotated rx 180 ry 0 rz -180 deg; joints [-31.037, 15.048, 63.216, 71.323, 32.973, -68.054]
  Call Extruder(271.64088)
  MoveL 8402 to (224.8, 164.7, 116.27) mm, rotated rx 180 ry 0 rz 180 deg; joints [-31.062, 14.991, 63.287, 71.361, 32.992, -68.093]
  MoveL 8403 to (224.8, 164.7, 116.27) mm, rotated rx 180 ry 0 rz 180 deg; joints [-31.062, 14.991, 63.287, 71.361, 32.992, -68.093]
  Call Extruder(271.83889)
  MoveL 8404 to (224.42, 164.75, 116.27) mm, rotated rx 180 ry 0 rz 180 deg; joints [-31.087, 14.934, 63.359, 71.399, 33.011, -68.132]
  MoveL 8405 to (224.42, 164.75, 116.27) mm, rotated rx 180 ry 0 rz 180 deg; joints [-31.087, 14.934, 63.359, 71.399, 33.011, -68.132]
  Call Extruder(272.03603)
  MoveL 8406 to (224.03, 164.79, 116.27) mm, rotated rx 180 ry 0 rz 180 deg; joints [-31.112, 14.877, 63.429, 71.437, 33.03, -68.171]
  MoveL 8407 to (224.03, 164.79, 116.27) mm, rotated rx 180 ry 0 rz 180 deg; joints [-31.112, 14.877, 63.429, 71.437, 33.03, -68.171]
  Call Extruder(272.23230)
  MoveL 8408 to (223.64, 164.84, 116.27) mm, rotated rx -180 ry 0 rz 180 deg; joints [-31.137, 14.82, 63.5, 71.474, 33.048, -68.21]
  MoveL 8409 to (223.64, 164.84, 116.27) mm, rotated rx -180 ry 0 rz 180 deg; joints [-31.137, 14.82, 63.5, 71.474, 33.048, -68.21]
  Call Extruder(272.47797)
  MoveL 8410 to (223.15, 164.89, 116.27) mm, rotated rx 180 ry 0 rz 180 deg; joints [-31.168, 14.748, 63.591, 71.521, 33.071, -68.258]
  MoveL 8411 to (223.15, 164.89, 116.27) mm, rotated rx 180 ry 0 rz 180 deg; joints [-31.168, 14.748, 63.591, 71.521, 33.071, -68.258]
  Call Extruder(272.77266)
  MoveL 8412 to (222.56, 164.93, 116.27) mm, rotated rx 180 ry 0 rz 180 deg; joints [-31.204, 14.659, 63.701, 71.577, 33.098, -68.317]
  MoveL 8413 to (222.56, 164.93, 116.27) mm, rotated rx 180 ry 0 rz 180 deg; joints [-31.204, 14.659, 63.701, 71.577, 33.098, -68.317]
  Call Extruder(273.06601)
  MoveL 8414 to (221.97, 164.98, 116.27) mm, rotated rx -180 ry 0 rz 180 deg; joints [-31.24, 14.571, 63.81, 71.633, 33.125, -68.374]
  MoveL 8415 to (221.97, 164.98, 116.27) mm, rotated rx -180 ry 0 rz 180 deg; joints [-31.24, 14.571, 63.81, 71.633, 33.125, -68.374]
  Call Extruder(273.49932)
  MoveL 8416 to (221.1, 165.03, 116.27) mm, rotated rx 180 ry 0 rz 180 deg; joints [-31.292, 14.438, 63.975, 71.715, 33.163, -68.459]
  MoveL 8417 to (221.1, 165.03, 116.27) mm, rotated rx 180 ry 0 rz 180 deg; joints [-31.292, 14.438, 63.975, 71.715, 33.163, -68.459]
  Call Extruder(274.07148)
  MoveL 8418 to (219.94, 165.07, 116.27) mm, rotated rx 180 ry 0 rz 180 deg; joints [-31.36, 14.261, 64.195, 71.821, 33.213, -68.571]
  MoveL 8419 to (219.94, 165.07, 116.27) mm, rotated rx 180 ry 0 rz 180 deg; joints [-31.36, 14.261, 64.195, 71.821, 33.213, -68.571]
  Call Extruder(274.49936)
  MoveL 8420 to (219.06, 165.09, 116.27) mm, rotated rx 180 ry 0 rz 180 deg; joints [-31.409, 14.126, 64.361, 71.9, 33.249, -68.653]
  Call Extruder(391.14801)
  MoveL 8421 to (-19.06, 165.09, 116.27) mm, rotated rx -180 ry 0 rz 180 deg; joints [-51.475, -14.579, 92.958, 80.889, 52.404, -75.273]
  MoveL 8422 to (-19.06, 165.09, 116.27) mm, rotated rx -180 ry 0 rz 180 deg; joints [-51.475, -14.579, 92.958, 80.889, 52.404, -75.273]
  Call Extruder(391.86364)
  MoveL 8423 to (-20.52, 165.05, 116.27) mm, rotated rx -180 ry 0 rz 180 deg; joints [-51.652, -14.715, 93.061, 80.921, 52.581, -75.266]
  MoveL 8424 to (-20.52, 165.05, 116.27) mm, rotated rx -180 ry 0 rz 180 deg; joints [-51.652, -14.715, 93.061, 80.921, 52.581, -75.266]
  Call Extruder(392.43838)
  MoveL 8425 to (-21.68, 165, 116.27) mm, rotated rx 180 ry 0 rz 180 deg; joints [-51.793, -14.824, 93.144, 80.946, 52.721, -75.26]
  MoveL 8426 to (-21.68, 165, 116.27) mm, rotated rx 180 ry 0 rz 180 deg; joints [-51.793, -14.824, 93.144, 80.946, 52.721, -75.26]
  Call Extruder(392.73174)
  MoveL 8427 to (-22.27, 164.96, 116.27) mm, rotated rx -180 ry 0 rz 180 deg; joints [-51.862, -14.882, 93.188, 80.957, 52.79, -75.255]
  MoveL 8428 to (-22.27, 164.96, 116.27) mm, rotated rx -180 ry 0 rz 180 deg; joints [-51.862, -14.882, 93.188, 80.957, 52.79, -75.255]
  Call Extruder(393.02643)
  MoveL 8429 to (-22.86, 164.91, 116.27) mm, rotated rx -180 ry 0 rz 180 deg; joints [-51.931, -14.94, 93.231, 80.968, 52.859, -75.251]
  MoveL 8430 to (-22.86, 164.91, 116.27) mm, rotated rx -180 ry 0 rz 180 deg; joints [-51.931, -14.94, 93.231, 80.968, 52.859, -75.251]
  Call Extruder(393.32246)
  MoveL 8431 to (-23.45, 164.86, 116.27) mm, rotated rx 180 ry 0 rz 180 deg; joints [-52.001, -14.998, 93.275, 80.98, 52.929, -75.246]
  MoveL 8432 to (-23.45, 164.86, 116.27) mm, rotated rx 180 ry 0 rz 180 deg; joints [-52.001, -14.998, 93.275, 80.98, 52.929, -75.246]
  Call Extruder(393.51873)
  MoveL 8433 to (-23.83, 164.82, 116.27) mm, rotated rx -180 ry 0 rz 180 deg; joints [-52.045, -15.038, 93.305, 80.986, 52.973, -75.243]
  MoveL 8434 to (-23.83, 164.82, 116.27) mm, rotated rx -180 ry 0 rz 180 deg; joints [-52.045, -15.038, 93.305, 80.986, 52.973, -75.243]
  Call Extruder(393.71587)
  MoveL 8435 to (-24.22, 164.77, 116.27) mm, rotated rx 180 ry 0 rz 180 deg; joints [-52.089, -15.078, 93.334, 80.993, 53.018, -75.239]
  MoveL 8436 to (-24.22, 164.77, 116.27) mm, rotated rx 180 ry 0 rz 180 deg; joints [-52.089, -15.078, 93.334, 80.993, 53.018, -75.239]
  Call Extruder(393.91388)
  MoveL 8437 to (-24.61, 164.73, 116.27) mm, rotated rx -180 ry 0 rz 180 deg; joints [-52.134, -15.118, 93.364, 81, 53.062, -75.235]
  MoveL 8438 to (-24.61, 164.73, 116.27) mm, rotated rx -180 ry 0 rz 180 deg; joints [-52.134, -15.118, 93.364, 81, 53.062, -75.235]
  Call Extruder(394.11275)
  MoveL 8439 to (-25, 164.68, 116.27) mm, rotated rx -180 ry 0 rz 180 deg; joints [-52.178, -15.157, 93.394, 81.007, 53.107, -75.231]
  MoveL 8440 to (-25, 164.68, 116.27) mm, rotated rx -180 ry 0 rz 180 deg; joints [-52.178, -15.157, 93.394, 81.007, 53.107, -75.231]
  Call Extruder(394.29183)
  MoveL 8441 to (-25.34, 164.63, 116.27) mm, rotated rx 180 ry 0 rz 180 deg; joints [-52.218, -15.194, 93.421, 81.012, 53.146, -75.227]
  MoveL 8442 to (-25.34, 164.63, 116.27) mm, rotated rx 180 ry 0 rz 180 deg; joints [-52.218, -15.194, 93.421, 81.012, 53.146, -75.227]
  Call Extruder(394.45103)
  MoveL 8443 to (-25.65, 164.58, 116.27) mm, rotated rx 180 ry 0 rz 180 deg; joints [-52.251, -15.226, 93.445, 81.017, 53.18, -75.224]
  MoveL 8444 to (-25.65, 164.58, 116.27) mm, rotated rx 180 ry 0 rz 180 deg; joints [-52.251, -15.226, 93.445, 81.017, 53.18, -75.224]
  Call Extruder(394.61095)
  MoveL 8445 to (-25.96, 164.54, 116.27) mm, rotated rx 180 ry 0 rz 180 deg; joints [-52.286, -15.259, 93.47, 81.022, 53.214, -75.22]
  MoveL 8446 to (-25.96, 164.54, 116.27) mm, rotated rx 180 ry 0 rz 180 deg; joints [-52.286, -15.259, 93.47, 81.022, 53.214, -75.22]
  Call Extruder(394.77161)
  MoveL 8447 to (-26.26, 164.49, 116.27) mm, rotated rx 180 ry 0 rz 180 deg; joints [-52.32, -15.292, 93.494, 81.027, 53.249, -75.216]
  MoveL 8448 to (-26.26, 164.49, 116.27) mm, rotated rx 180 ry 0 rz 180 deg; joints [-52.32, -15.292, 93.494, 81.027, 53.249, -75.216]
  Call Extruder(394.93299)
  MoveL 8449 to (-26.57, 164.44, 116.27) mm, rotated rx 180 ry 0 rz -180 deg; joints [-52.354, -15.324, 93.518, 81.031, 53.283, -75.212]
  MoveL 8450 to (-26.57, 164.44, 116.27) mm, rotated rx 180 ry 0 rz -180 deg; joints [-52.354, -15.324, 93.518, 81.031, 53.283, -75.212]
  Call Extruder(395.09509)
  MoveL 8451 to (-26.87, 164.39, 116.27) mm, rotated rx -180 ry 0 rz 180 deg; joints [-52.388, -15.357, 93.543, 81.036, 53.317, -75.209]
  MoveL 8452 to (-26.87, 164.39, 116.27) mm, rotated rx -180 ry 0 rz 180 deg; joints [-52.388, -15.357, 93.543, 81.036, 53.317, -75.209]
  Call Extruder(395.24330)
  MoveL 8453 to (-27.15, 164.34, 116.27) mm, rotated rx -180 ry 0 rz 180 deg; joints [-52.418, -15.387, 93.565, 81.04, 53.348, -75.205]
  MoveL 8454 to (-27.15, 164.34, 116.27) mm, rotated rx -180 ry 0 rz 180 deg; joints [-52.418, -15.387, 93.565, 81.04, 53.348, -75.205]
  Call Extruder(395.37753)
  MoveL 8455 to (-27.4, 164.29, 116.27) mm, rotated rx 180 ry 0 rz 180 deg; joints [-52.445, -15.415, 93.586, 81.043, 53.375, -75.201]
  MoveL 8456 to (-27.4, 164.29, 116.27) mm, rotated rx 180 ry 0 rz 180 deg; joints [-52.445, -15.415, 93.586, 81.043, 53.375, -75.201]
  Call Extruder(395.51237)
  MoveL 8457 to (-27.65, 164.24, 116.27) mm, rotated rx 180 ry 0 rz 180 deg; joints [-52.472, -15.442, 93.606, 81.047, 53.402, -75.198]
  MoveL 8458 to (-27.65, 164.24, 116.27) mm, rotated rx 180 ry 0 rz 180 deg; joints [-52.472, -15.442, 93.606, 81.047, 53.402, -75.198]
  Call Extruder(395.64782)
  MoveL 8459 to (-27.9, 164.19, 116.27) mm, rotated rx 180 ry 0 rz 180 deg; joints [-52.499, -15.47, 93.627, 81.05, 53.429, -75.194]
  MoveL 8460 to (-27.9, 164.19, 116.27) mm, rotated rx 180 ry 0 rz 180 deg; joints [-52.499, -15.47, 93.627, 81.05, 53.429, -75.194]
  Call Extruder(395.78388)
  MoveL 8461 to (-28.15, 164.14, 116.27) mm, rotated rx 180 ry 0 rz -180 deg; joints [-52.526, -15.498, 93.647, 81.053, 53.457, -75.19]
  MoveL 8462 to (-28.15, 164.14, 116.27) mm, rotated rx 180 ry 0 rz -180 deg; joints [-52.526, -15.498, 93.647, 81.053, 53.457, -75.19]
  Call Extruder(395.92056)
  MoveL 8463 to (-28.4, 164.09, 116.27) mm, rotated rx 180 ry 0 rz 180 deg; joints [-52.553, -15.525, 93.668, 81.057, 53.484, -75.187]
  MoveL 8464 to (-28.4, 164.09, 116.27) mm, rotated rx 180 ry 0 rz 180 deg; joints [-52.553, -15.525, 93.668, 81.057, 53.484, -75.187]
  Call Extruder(396.05784)
  MoveL 8465 to (-28.64, 164.04, 116.27) mm, rotated rx -180 ry 0 rz 180 deg; joints [-52.58, -15.553, 93.688, 81.06, 53.511, -75.183]
  MoveL 8466 to (-28.64, 164.04, 116.27) mm, rotated rx -180 ry 0 rz 180 deg; joints [-52.58, -15.553, 93.688, 81.06, 53.511, -75.183]
  Call Extruder(396.18351)
  MoveL 8467 to (-28.87, 164, 116.27) mm, rotated rx 180 ry 0 rz 180 deg; joints [-52.605, -15.578, 93.707, 81.063, 53.536, -75.18]
  MoveL 8468 to (-28.87, 164, 116.27) mm, rotated rx 180 ry 0 rz 180 deg; joints [-52.605, -15.578, 93.707, 81.063, 53.536, -75.18]
  Call Extruder(396.29745)
  MoveL 8469 to (-29.08, 163.95, 116.27) mm, rotated rx -180 ry 0 rz 180 deg; joints [-52.627, -15.601, 93.724, 81.066, 53.558, -75.176]
  MoveL 8470 to (-29.08, 163.95, 116.27) mm, rotated rx -180 ry 0 rz 180 deg; joints [-52.627, -15.601, 93.724, 81.066, 53.558, -75.176]
  Call Extruder(396.41184)
  MoveL 8471 to (-29.28, 163.91, 116.27) mm, rotated rx 180 ry 0 rz 180 deg; joints [-52.649, -15.624, 93.741, 81.068, 53.58, -75.173]
  MoveL 8472 to (-29.28, 163.91, 116.27) mm, rotated rx 180 ry 0 rz 180 deg; joints [-52.649, -15.624, 93.741, 81.068, 53.58, -75.173]
  Call Extruder(396.52669)
  MoveL 8473 to (-29.48, 163.86, 116.27) mm, rotated rx -180 ry 0 rz 180 deg; joints [-52.67, -15.647, 93.758, 81.071, 53.602, -75.17]
  MoveL 8474 to (-29.48, 163.86, 116.27) mm, rotated rx -180 ry 0 rz 180 deg; joints [-52.67, -15.647, 93.758, 81.071, 53.602, -75.17]
  Call Extruder(396.64199)
  MoveL 8475 to (-29.69, 163.82, 116.27) mm, rotated rx -180 ry 0 rz 180 deg; joints [-52.692, -15.67, 93.775, 81.074, 53.624, -75.167]
  MoveL 8476 to (-29.69, 163.82, 116.27) mm, rotated rx -180 ry 0 rz 180 deg; joints [-52.692, -15.67, 93.775, 81.074, 53.624, -75.167]
  Call Extruder(396.77138)
  MoveL 8477 to (-29.91, 163.75, 116.27) mm, rotated rx 180 ry 0 rz 180 deg; joints [-52.714, -15.698, 93.795, 81.075, 53.647, -75.162]
  MoveL 8478 to (-29.91, 163.75, 116.27) mm, rotated rx 180 ry 0 rz 180 deg; joints [-52.714, -15.698, 93.795, 81.075, 53.647, -75.162]
  Call Extruder(396.90134)
  MoveL 8479 to (-30.14, 163.68, 116.27) mm, rotated rx 180 ry 0 rz 180 deg; joints [-52.737, -15.725, 93.816, 81.077, 53.669, -75.157]
  MoveL 8480 to (-30.14, 163.68, 116.27) mm, rotated rx 180 ry 0 rz 180 deg; joints [-52.737, -15.725, 93.816, 81.077, 53.669, -75.157]
  Call Extruder(397.03187)
  MoveL 8481 to (-30.36, 163.62, 116.27) mm, rotated rx 180 ry 0 rz 180 deg; joints [-52.759, -15.752, 93.836, 81.079, 53.692, -75.153]
  MoveL 8482 to (-30.36, 163.62, 116.27) mm, rotated rx 180 ry 0 rz 180 deg; joints [-52.759, -15.752, 93.836, 81.079, 53.692, -75.153]
  Call Extruder(397.16296)
  MoveL 8483 to (-30.58, 163.55, 116.27) mm, rotated rx 180 ry 0 rz 180 deg; joints [-52.781, -15.78, 93.856, 81.081, 53.714, -75.148]
  MoveL 8484 to (-30.58, 163.55, 116.27) mm, rotated rx 180 ry 0 rz 180 deg; joints [-52.781, -15.78, 93.856, 81.081, 53.714, -75.148]
  Call Extruder(397.28461)
  MoveL 8485 to (-30.79, 163.48, 116.27) mm, rotated rx -180 ry 0 rz 180 deg; joints [-52.801, -15.805, 93.875, 81.083, 53.735, -75.144]
  MoveL 8486 to (-30.79, 163.48, 116.27) mm, rotated rx -180 ry 0 rz 180 deg; joints [-52.801, -15.805, 93.875, 81.083, 53.735, -75.144]
  Call Extruder(397.39672)
  MoveL 8487 to (-30.98, 163.42, 116.27) mm, rotated rx 180 ry 0 rz 180 deg; joints [-52.82, -15.829, 93.892, 81.084, 53.754, -75.14]
  MoveL 8488 to (-30.98, 163.42, 116.27) mm, rotated rx 180 ry 0 rz 180 deg; joints [-52.82, -15.829, 93.892, 81.084, 53.754, -75.14]
  Call Extruder(397.50928)
  MoveL 8489 to (-31.17, 163.36, 116.27) mm, rotated rx 180 ry 0 rz 180 deg; joints [-52.838, -15.852, 93.909, 81.085, 53.772, -75.136]
  MoveL 8490 to (-31.17, 163.36, 116.27) mm, rotated rx 180 ry 0 rz 180 deg; joints [-52.838, -15.852, 93.909, 81.085, 53.772, -75.136]
  Call Extruder(397.54120)
  MoveL 8491 to (-31.22, 163.34, 116.27) mm, rotated rx 180 ry 0 rz 180 deg; joints [-52.843, -15.859, 93.914, 81.086, 53.778, -75.134]
  Set speed (130.0 mm/s)
  MoveL 8492 to (-34.34, 162.18, 116.27) mm, rotated rx 180 ry 0 rz 180 deg; joints [-53.135, -16.264, 94.211, 81.1, 54.077, -75.056]
  MoveL 8493 to (-34.34, 162.18, 125.68) mm, rotated rx 180 ry 0 rz 180 deg; joints [-53.135, -16.869, 96.071, 82.003, 53.892, -76.592]
  MoveL 8494 to (-31.64, 163.21, 125.68) mm, rotated rx -180 ry 0 rz 180 deg; joints [-52.884, -16.513, 95.813, 82.002, 53.634, -76.669]
  Set speed (30.0 mm/s)
  MoveL 8495 to (-31.64, 163.21, 125.68) mm, rotated rx -180 ry 0 rz 180 deg; joints [-52.884, -16.513, 95.813, 82.002, 53.634, -76.669]
  Call Extruder(397.72317)
  MoveL 8496 to (-31.93, 163.09, 125.68) mm, rotated rx -180 ry 0 rz 180 deg; joints [-52.91, -16.553, 95.842, 82.002, 53.661, -76.66]
  MoveL 8497 to (-31.93, 163.09, 125.68) mm, rotated rx -180 ry 0 rz 180 deg; joints [-52.91, -16.553, 95.842, 82.002, 53.661, -76.66]
  Call Extruder(397.90591)
  MoveL 8498 to (-32.22, 162.97, 125.68) mm, rotated rx 180 ry 0 rz 180 deg; joints [-52.936, -16.593, 95.871, 82.001, 53.688, -76.651]
  MoveL 8499 to (-32.22, 162.97, 125.68) mm, rotated rx 180 ry 0 rz 180 deg; joints [-52.936, -16.593, 95.871, 82.001, 53.688, -76.651]
  Call Extruder(398.07632)
  MoveL 8500 to (-32.49, 162.85, 125.68) mm, rotated rx 180 ry 0 rz 180 deg; joints [-52.96, -16.629, 95.898, 82.001, 53.713, -76.643]
  MoveL 8501 to (-32.49, 162.85, 125.68) mm, rotated rx 180 ry 0 rz 180 deg; joints [-52.96, -16.629, 95.898, 82.001, 53.713, -76.643]
  Call Extruder(398.23430)
  MoveL 8502 to (-32.74, 162.74, 125.68) mm, rotated rx 180 ry 0 rz 180 deg; joints [-52.982, -16.664, 95.923, 82, 53.735, -76.635]
  MoveL 8503 to (-32.74, 162.74, 125.68) mm, rotated rx 180 ry 0 rz 180 deg; joints [-52.982, -16.664, 95.923, 82, 53.735, -76.635]
  Call Extruder(398.39287)
  MoveL 8504 to (-32.99, 162.64, 125.68) mm, rotated rx 180 ry 0 rz 180 deg; joints [-53.004, -16.698, 95.947, 82, 53.758, -76.627]
  MoveL 8505 to (-32.99, 162.64, 125.68) mm, rotated rx 180 ry 0 rz 180 deg; joints [-53.004, -16.698, 95.947, 82, 53.758, -76.627]
  Call Extruder(398.59904)
  MoveL 8506 to (-33.29, 162.46, 125.68) mm, rotated rx -180 ry 0 rz 180 deg; joints [-53.026, -16.745, 95.981, 81.997, 53.782, -76.615]
  MoveL 8507 to (-33.29, 162.46, 125.68) mm, rotated rx -180 ry 0 rz 180 deg; joints [-53.026, -16.745, 95.981, 81.997, 53.782, -76.615]
  Call Extruder(398.80598)
  MoveL 8508 to (-33.6, 162.29, 125.68) mm, rotated rx -180 ry 0 rz 180 deg; joints [-53.049, -16.792, 96.015, 81.994, 53.805, -76.603]
  MoveL 8509 to (-33.6, 162.29, 125.68) mm, rotated rx -180 ry 0 rz 180 deg; joints [-53.049, -16.792, 96.015, 81.994, 53.805, -76.603]
  Call Extruder(399.01371)
  MoveL 8510 to (-33.9, 162.11, 125.68) mm, rotated rx 180 ry 0 rz 180 deg; joints [-53.071, -16.838, 96.049, 81.991, 53.829, -76.591]
  MoveL 8511 to (-33.9, 162.11, 125.68) mm, rotated rx 180 ry 0 rz 180 deg; joints [-53.071, -16.838, 96.049, 81.991, 53.829, -76.591]
  Call Extruder(399.22221)
  MoveL 8512 to (-34.21, 161.93, 125.68) mm, rotated rx 180 ry 0 rz 180 deg; joints [-53.094, -16.885, 96.083, 81.988, 53.853, -76.579]
  MoveL 8513 to (-34.21, 161.93, 125.68) mm, rotated rx 180 ry 0 rz 180 deg; joints [-53.094, -16.885, 96.083, 81.988, 53.853, -76.579]
  Call Extruder(399.40175)
  MoveL 8514 to (-34.45, 161.76, 125.68) mm, rotated rx 180 ry 0 rz 180 deg; joints [-53.109, -16.927, 96.113, 81.984, 53.869, -76.567]
  MoveL 8515 to (-34.45, 161.76, 125.68) mm, rotated rx 180 ry 0 rz 180 deg; joints [-53.109, -16.927, 96.113, 81.984, 53.869, -76.567]
  Call Extruder(399.73518)
  MoveL 8516 to (-34.9, 161.43, 125.68) mm, rotated rx -180 ry 0 rz -180 deg; joints [-53.135, -17.004, 96.169, 81.976, 53.898, -76.545]
  MoveL 8517 to (-34.9, 161.43, 125.68) mm, rotated rx -180 ry 0 rz -180 deg; joints [-53.135, -17.004, 96.169, 81.976, 53.898, -76.545]
  Call Extruder(400.06980)
  MoveL 8518 to (-35.35, 161.1, 125.68) mm, rotated rx -180 ry 0 rz -180 deg; joints [-53.163, -17.082, 96.224, 81.968, 53.927, -76.523]
  Call Extruder(400.89771)
  MoveL 8519 to (-36.39, 160.19, 125.68) mm, rotated rx -180 ry 0 rz -180 deg; joints [-53.209, -17.278, 96.365, 81.942, 53.98, -76.463]
  Call Extruder(401.72565)
  MoveL 8520 to (-37.3, 159.15, 125.68) mm, rotated rx 180 ry 0 rz -180 deg; joints [-53.227, -17.477, 96.507, 81.906, 54.006, -76.397]
  Call Extruder(401.89295)
  MoveL 8521 to (-37.47, 158.93, 125.68) mm, rotated rx -180 ry 0 rz -180 deg; joints [-53.227, -17.517, 96.536, 81.897, 54.007, -76.382]
  MoveL 8522 to (-37.47, 158.93, 125.68) mm, rotated rx -180 ry 0 rz -180 deg; joints [-53.227, -17.517, 96.536, 81.897, 54.007, -76.382]
  Call Extruder(402.22638)
  MoveL 8523 to (-37.8, 158.48, 125.68) mm, rotated rx 180 ry 0 rz -180 deg; joints [-53.226, -17.598, 96.593, 81.88, 54.009, -76.353]
  MoveL 8524 to (-37.8, 158.48, 125.68) mm, rotated rx 180 ry 0 rz -180 deg; joints [-53.226, -17.598, 96.593, 81.88, 54.009, -76.353]
  Call Extruder(402.55863)
  MoveL 8525 to (-38.12, 158.03, 125.68) mm, rotated rx -180 ry 0 rz 180 deg; joints [-53.224, -17.679, 96.65, 81.863, 54.011, -76.324]
  MoveL 8526 to (-38.12, 158.03, 125.68) mm, rotated rx -180 ry 0 rz 180 deg; joints [-53.224, -17.679, 96.65, 81.863, 54.011, -76.324]
  Call Extruder(402.67630)
  MoveL 8527 to (-38.22, 157.85, 125.68) mm, rotated rx -180 ry 0 rz 180 deg; joints [-53.221, -17.707, 96.67, 81.856, 54.009, -76.314]
  MoveL 8528 to (-38.22, 157.85, 125.68) mm, rotated rx -180 ry 0 rz 180 deg; joints [-53.221, -17.707, 96.67, 81.856, 54.009, -76.314]
  Call Extruder(402.88403)
  MoveL 8529 to (-38.4, 157.55, 125.68) mm, rotated rx 180 ry 0 rz 180 deg; joints [-53.214, -17.758, 96.706, 81.843, 54.004, -76.294]
  MoveL 8530 to (-38.4, 157.55, 125.68) mm, rotated rx 180 ry 0 rz 180 deg; joints [-53.214, -17.758, 96.706, 81.843, 54.004, -76.294]
  Call Extruder(403.09097)
  MoveL 8531 to (-38.57, 157.25, 125.68) mm, rotated rx 180 ry 0 rz 180 deg; joints [-53.207, -17.808, 96.742, 81.83, 53.999, -76.275]
  MoveL 8532 to (-38.57, 157.25, 125.68) mm, rotated rx 180 ry 0 rz 180 deg; joints [-53.207, -17.808, 96.742, 81.83, 53.999, -76.275]
  Call Extruder(403.29714)
  MoveL 8533 to (-38.75, 156.94, 125.68) mm, rotated rx 180 ry 0 rz 180 deg; joints [-53.2, -17.858, 96.777, 81.818, 53.995, -76.256]
  MoveL 8534 to (-38.75, 156.94, 125.68) mm, rotated rx 180 ry 0 rz 180 deg; joints [-53.2, -17.858, 96.777, 81.818, 53.995, -76.256]
  Call Extruder(403.47882)
  MoveL 8535 to (-38.89, 156.66, 125.68) mm, rotated rx 180 ry 0 rz 180 deg; joints [-53.191, -17.903, 96.809, 81.806, 53.988, -76.238]
  MoveL 8536 to (-38.89, 156.66, 125.68) mm, rotated rx 180 ry 0 rz 180 deg; joints [-53.191, -17.903, 96.809, 81.806, 53.988, -76.238]
  Call Extruder(403.63681)
  MoveL 8537 to (-39, 156.42, 125.68) mm, rotated rx 180 ry 0 rz 180 deg; joints [-53.18, -17.941, 96.835, 81.795, 53.979, -76.223]
  MoveL 8538 to (-39, 156.42, 125.68) mm, rotated rx 180 ry 0 rz 180 deg; joints [-53.18, -17.941, 96.835, 81.795, 53.979, -76.223]
  Call Extruder(403.79419)
  MoveL 8539 to (-39.11, 156.17, 125.68) mm, rotated rx 180 ry 0 rz 180 deg; joints [-53.17, -17.979, 96.862, 81.783, 53.971, -76.207]
  MoveL 8540 to (-39.11, 156.17, 125.68) mm, rotated rx 180 ry 0 rz 180 deg; joints [-53.17, -17.979, 96.862, 81.783, 53.971, -76.207]
  Call Extruder(403.97691)
  MoveL 8541 to (-39.23, 155.87, 125.68) mm, rotated rx 180 ry 0 rz 180 deg; joints [-53.156, -18.023, 96.893, 81.77, 53.96, -76.189]
  MoveL 8542 to (-39.23, 155.87, 125.68) mm, rotated rx 180 ry 0 rz 180 deg; joints [-53.156, -18.023, 96.893, 81.77, 53.96, -76.189]
  Call Extruder(404.15887)
  MoveL 8543 to (-39.35, 155.58, 125.68) mm, rotated rx 180 ry 0 rz 180 deg; joints [-53.143, -18.067, 96.924, 81.757, 53.949, -76.17]
  MoveL 8544 to (-39.35, 155.58, 125.68) mm, rotated rx 180 ry 0 rz 180 deg; joints [-53.143, -18.067, 96.924, 81.757, 53.949, -76.17]
  Call Extruder(404.30621)
  MoveL 8545 to (-39.44, 155.34, 125.68) mm, rotated rx 180 ry 0 rz -180 deg; joints [-53.131, -18.103, 96.949, 81.745, 53.939, -76.155]
  MoveL 8546 to (-39.44, 155.34, 125.68) mm, rotated rx 180 ry 0 rz -180 deg; joints [-53.131, -18.103, 96.949, 81.745, 53.939, -76.155]
  Call Extruder(404.41944)
  MoveL 8547 to (-39.5, 155.15, 125.68) mm, rotated rx -180 ry 0 rz 180 deg; joints [-53.121, -18.13, 96.968, 81.736, 53.93, -76.143]
  MoveL 8548 to (-39.5, 155.15, 125.68) mm, rotated rx -180 ry 0 rz 180 deg; joints [-53.121, -18.13, 96.968, 81.736, 53.93, -76.143]
  Call Extruder(404.53223)
  MoveL 8549 to (-39.56, 154.97, 125.68) mm, rotated rx 180 ry 0 rz 180 deg; joints [-53.11, -18.157, 96.987, 81.727, 53.92, -76.132]
  MoveL 8550 to (-39.56, 154.97, 125.68) mm, rotated rx 180 ry 0 rz 180 deg; joints [-53.11, -18.157, 96.987, 81.727, 53.92, -76.132]
  Call Extruder(404.64458)
  MoveL 8551 to (-39.62, 154.78, 125.68) mm, rotated rx -180 ry 0 rz 180 deg; joints [-53.099, -18.184, 97.006, 81.718, 53.911, -76.12]
  MoveL 8552 to (-39.62, 154.78, 125.68) mm, rotated rx -180 ry 0 rz 180 deg; joints [-53.099, -18.184, 97.006, 81.718, 53.911, -76.12]
  Call Extruder(404.75648)
  MoveL 8553 to (-39.68, 154.59, 125.68) mm, rotated rx 180 ry 0 rz -180 deg; joints [-53.088, -18.211, 97.025, 81.709, 53.902, -76.108]
  MoveL 8554 to (-39.68, 154.59, 125.68) mm, rotated rx 180 ry 0 rz -180 deg; joints [-53.088, -18.211, 97.025, 81.709, 53.902, -76.108]
  Call Extruder(404.87788)
  MoveL 8555 to (-39.75, 154.38, 125.68) mm, rotated rx 180 ry 0 rz -180 deg; joints [-53.076, -18.241, 97.046, 81.699, 53.891, -76.095]
  MoveL 8556 to (-39.75, 154.38, 125.68) mm, rotated rx 180 ry 0 rz -180 deg; joints [-53.076, -18.241, 97.046, 81.699, 53.891, -76.095]
  Call Extruder(405.00867)
  MoveL 8557 to (-39.81, 154.16, 125.68) mm, rotated rx 180 ry 0 rz 180 deg; joints [-53.063, -18.273, 97.068, 81.688, 53.879, -76.081]
  MoveL 8558 to (-39.81, 154.16, 125.68) mm, rotated rx 180 ry 0 rz 180 deg; joints [-53.063, -18.273, 97.068, 81.688, 53.879, -76.081]
  Call Extruder(405.13890)
  MoveL 8559 to (-39.88, 153.94, 125.68) mm, rotated rx 180 ry 0 rz 180 deg; joints [-53.049, -18.304, 97.09, 81.677, 53.868, -76.067]
  MoveL 8560 to (-39.88, 153.94, 125.68) mm, rotated rx 180 ry 0 rz 180 deg; joints [-53.049, -18.304, 97.09, 81.677, 53.868, -76.067]
  Call Extruder(405.26856)
  MoveL 8561 to (-39.95, 153.71, 125.68) mm, rotated rx 180 ry 0 rz 180 deg; joints [-53.036, -18.336, 97.112, 81.667, 53.856, -76.053]
  MoveL 8562 to (-39.95, 153.71, 125.68) mm, rotated rx 180 ry 0 rz 180 deg; joints [-53.036, -18.336, 97.112, 81.667, 53.856, -76.053]
  Call Extruder(405.39766)
  MoveL 8563 to (-40.02, 153.49, 125.68) mm, rotated rx 180 ry 0 rz 180 deg; joints [-53.022, -18.367, 97.134, 81.656, 53.844, -76.039]
  MoveL 8564 to (-40.02, 153.49, 125.68) mm, rotated rx 180 ry 0 rz 180 deg; joints [-53.022, -18.367, 97.134, 81.656, 53.844, -76.039]
  Call Extruder(405.51275)
  MoveL 8565 to (-40.06, 153.28, 125.68) mm, rotated rx 180 ry 0 rz -180 deg; joints [-53.007, -18.395, 97.153, 81.645, 53.831, -76.026]
  MoveL 8566 to (-40.06, 153.28, 125.68) mm, rotated rx 180 ry 0 rz -180 deg; joints [-53.007, -18.395, 97.153, 81.645, 53.831, -76.026]
  Call Extruder(405.62739)
  MoveL 8567 to (-40.11, 153.08, 125.68) mm, rotated rx 180 ry 0 rz 180 deg; joints [-52.993, -18.422, 97.172, 81.635, 53.818, -76.013]
  MoveL 8568 to (-40.11, 153.08, 125.68) mm, rotated rx 180 ry 0 rz 180 deg; joints [-52.993, -18.422, 97.172, 81.635, 53.818, -76.013]
  Call Extruder(405.74157)
  MoveL 8569 to (-40.15, 152.88, 125.68) mm, rotated rx 180 ry 0 rz 180 deg; joints [-52.978, -18.45, 97.191, 81.624, 53.805, -76]
  MoveL 8570 to (-40.15, 152.88, 125.68) mm, rotated rx 180 ry 0 rz 180 deg; joints [-52.978, -18.45, 97.191, 81.624, 53.805, -76]
  Call Extruder(405.85530)
  MoveL 8571 to (-40.2, 152.67, 125.68) mm, rotated rx 180 ry 0 rz -180 deg; joints [-52.963, -18.477, 97.211, 81.614, 53.792, -75.987]
  MoveL 8572 to (-40.2, 152.67, 125.68) mm, rotated rx 180 ry 0 rz -180 deg; joints [-52.963, -18.477, 97.211, 81.614, 53.792, -75.987]
  Call Extruder(405.98072)
  MoveL 8573 to (-40.24, 152.45, 125.68) mm, rotated rx 180 ry 0 rz 180 deg; joints [-52.946, -18.507, 97.232, 81.602, 53.777, -75.973]
  MoveL 8574 to (-40.24, 152.45, 125.68) mm, rotated rx 180 ry 0 rz 180 deg; joints [-52.946, -18.507, 97.232, 81.602, 53.777, -75.973]
  Call Extruder(406.11770)
  MoveL 8575 to (-40.29, 152.2, 125.68) mm, rotated rx -180 ry 0 rz 180 deg; joints [-52.928, -18.54, 97.254, 81.589, 53.76, -75.958]
  MoveL 8576 to (-40.29, 152.2, 125.68) mm, rotated rx -180 ry 0 rz 180 deg; joints [-52.928, -18.54, 97.254, 81.589, 53.76, -75.958]
  Call Extruder(406.25406)
  MoveL 8577 to (-40.34, 151.95, 125.68) mm, rotated rx 180 ry 0 rz 180 deg; joints [-52.909, -18.573, 97.277, 81.576, 53.743, -75.942]
  MoveL 8578 to (-40.34, 151.95, 125.68) mm, rotated rx 180 ry 0 rz 180 deg; joints [-52.909, -18.573, 97.277, 81.576, 53.743, -75.942]
  Call Extruder(406.38982)
  MoveL 8579 to (-40.39, 151.7, 125.68) mm, rotated rx 180 ry 0 rz 180 deg; joints [-52.89, -18.606, 97.3, 81.563, 53.727, -75.926]
  MoveL 8580 to (-40.39, 151.7, 125.68) mm, rotated rx 180 ry 0 rz 180 deg; joints [-52.89, -18.606, 97.3, 81.563, 53.727, -75.926]
  Call Extruder(406.52496)
  MoveL 8581 to (-40.44, 151.45, 125.68) mm, rotated rx 180 ry 0 rz 180 deg; joints [-52.871, -18.639, 97.323, 81.55, 53.71, -75.91]
  MoveL 8582 to (-40.44, 151.45, 125.68) mm, rotated rx 180 ry 0 rz 180 deg; joints [-52.871, -18.639, 97.323, 81.55, 53.71, -75.91]
  Call Extruder(406.65950)
  MoveL 8583 to (-40.49, 151.2, 125.68) mm, rotated rx 180 ry 0 rz 180 deg; joints [-52.853, -18.672, 97.346, 81.537, 53.693, -75.894]
  MoveL 8584 to (-40.49, 151.2, 125.68) mm, rotated rx 180 ry 0 rz 180 deg; joints [-52.853, -18.672, 97.346, 81.537, 53.693, -75.894]
  Call Extruder(406.79342)
  MoveL 8585 to (-40.54, 150.95, 125.68) mm, rotated rx 180 ry 0 rz 180 deg; joints [-52.834, -18.705, 97.369, 81.524, 53.676, -75.879]
  MoveL 8586 to (-40.54, 150.95, 125.68) mm, rotated rx 180 ry 0 rz 180 deg; joints [-52.834, -18.705, 97.369, 81.524, 53.676, -75.879]
  Call Extruder(406.94128)
  MoveL 8587 to (-40.59, 150.67, 125.68) mm, rotated rx -180 ry 0 rz 180 deg; joints [-52.812, -18.741, 97.394, 81.509, 53.657, -75.861]
  MoveL 8588 to (-40.59, 150.67, 125.68) mm, rotated rx -180 ry 0 rz 180 deg; joints [-52.812, -18.741, 97.394, 81.509, 53.657, -75.861]
  Call Extruder(407.10301)
  MoveL 8589 to (-40.64, 150.37, 125.68) mm, rotated rx -180 ry 0 rz 180 deg; joints [-52.787, -18.78, 97.421, 81.493, 53.635, -75.842]
  MoveL 8590 to (-40.64, 150.37, 125.68) mm, rotated rx -180 ry 0 rz 180 deg; joints [-52.787, -18.78, 97.421, 81.493, 53.635, -75.842]
  Call Extruder(407.26400)
  MoveL 8591 to (-40.69, 150.06, 125.68) mm, rotated rx 180 ry 0 rz 180 deg; joints [-52.762, -18.82, 97.448, 81.476, 53.612, -75.822]
  MoveL 8592 to (-40.69, 150.06, 125.68) mm, rotated rx 180 ry 0 rz 180 deg; joints [-52.762, -18.82, 97.448, 81.476, 53.612, -75.822]
  Call Extruder(407.42427)
  MoveL 8593 to (-40.73, 149.76, 125.68) mm, rotated rx 180 ry 0 rz 180 deg; joints [-52.737, -18.859, 97.475, 81.46, 53.59, -75.803]
  MoveL 8594 to (-40.73, 149.76, 125.68) mm, rotated rx 180 ry 0 rz 180 deg; joints [-52.737, -18.859, 97.475, 81.46, 53.59, -75.803]
  Call Extruder(407.58382)
  MoveL 8595 to (-40.78, 149.45, 125.68) mm, rotated rx 180 ry 0 rz 180 deg; joints [-52.712, -18.898, 97.502, 81.443, 53.567, -75.783]
  MoveL 8596 to (-40.78, 149.45, 125.68) mm, rotated rx 180 ry 0 rz 180 deg; joints [-52.712, -18.898, 97.502, 81.443, 53.567, -75.783]
  Call Extruder(407.74263)
  MoveL 8597 to (-40.83, 149.14, 125.68) mm, rotated rx 180 ry 0 rz 180 deg; joints [-52.687, -18.938, 97.529, 81.427, 53.545, -75.763]
  MoveL 8598 to (-40.83, 149.14, 125.68) mm, rotated rx 180 ry 0 rz 180 deg; joints [-52.687, -18.938, 97.529, 81.427, 53.545, -75.763]
  Call Extruder(407.92129)
  MoveL 8599 to (-40.88, 148.8, 125.68) mm, rotated rx 180 ry 0 rz 180 deg; joints [-52.658, -18.981, 97.559, 81.408, 53.519, -75.741]
  MoveL 8600 to (-40.88, 148.8, 125.68) mm, rotated rx 180 ry 0 rz 180 deg; joints [-52.658, -18.981, 97.559, 81.408, 53.519, -75.741]
  Call Extruder(408.11974)
  MoveL 8601 to (-40.93, 148.41, 125.68) mm, rotated rx 180 ry 0 rz 180 deg; joints [-52.624, -19.03, 97.592, 81.386, 53.488, -75.716]
  MoveL 8602 to (-40.93, 148.41, 125.68) mm, rotated rx 180 ry 0 rz 180 deg; joints [-52.624, -19.03, 97.592, 81.386, 53.488, -75.716]
  Call Extruder(408.31731)
  MoveL 8603 to (-40.97, 148.02, 125.68) mm, rotated rx 180 ry 0 rz 180 deg; joints [-52.59, -19.078, 97.625, 81.365, 53.457, -75.692]
  MoveL 8604 to (-40.97, 148.02, 125.68) mm, rotated rx 180 ry 0 rz 180 deg; joints [-52.59, -19.078, 97.625, 81.365, 53.457, -75.692]
  Call Extruder(408.51402)
  MoveL 8605 to (-41.02, 147.63, 125.68) mm, rotated rx -180 ry 0 rz -180 deg; joints [-52.556, -19.126, 97.659, 81.343, 53.427, -75.667]
  MoveL 8606 to (-41.02, 147.63, 125.68) mm, rotated rx -180 ry 0 rz -180 deg; joints [-52.556, -19.126, 97.659, 81.343, 53.427, -75.667]
  Call Extruder(408.70985)
  MoveL 8607 to (-41.06, 147.25, 125.68) mm, rotated rx 180 ry 0 rz 180 deg; joints [-52.521, -19.175, 97.691, 81.321, 53.396, -75.641]
  MoveL 8608 to (-41.06, 147.25, 125.68) mm, rotated rx 180 ry 0 rz 180 deg; joints [-52.521, -19.175, 97.691, 81.321, 53.396, -75.641]
  Call Extruder(409.00525)
  MoveL 8609 to (-41.11, 146.66, 125.68) mm, rotated rx 180 ry 0 rz 180 deg; joints [-52.466, -19.246, 97.74, 81.288, 53.346, -75.603]
  MoveL 8610 to (-41.11, 146.66, 125.68) mm, rotated rx 180 ry 0 rz 180 deg; joints [-52.466, -19.246, 97.74, 81.288, 53.346, -75.603]
  Call Extruder(409.29932)
  MoveL 8611 to (-41.16, 146.07, 125.68) mm, rotated rx 180 ry 0 rz 180 deg; joints [-52.411, -19.317, 97.789, 81.254, 53.295, -75.565]
  MoveL 8612 to (-41.16, 146.07, 125.68) mm, rotated rx 180 ry 0 rz 180 deg; joints [-52.411, -19.317, 97.789, 81.254, 53.295, -75.565]
  Call Extruder(409.59205)
  MoveL 8613 to (-41.2, 145.48, 125.68) mm, rotated rx 180 ry 0 rz 180 deg; joints [-52.355, -19.389, 97.837, 81.22, 53.245, -75.527]
  MoveL 8614 to (-41.2, 145.48, 125.68) mm, rotated rx 180 ry 0 rz 180 deg; joints [-52.355, -19.389, 97.837, 81.22, 53.245, -75.527]
  Call Extruder(410.16551)
  MoveL 8615 to (-41.25, 144.32, 125.68) mm, rotated rx 180 ry 0 rz -180 deg; joints [-52.239, -19.525, 97.93, 81.151, 53.139, -75.451]
  MoveL 8616 to (-41.25, 144.32, 125.68) mm, rotated rx 180 ry 0 rz -180 deg; joints [-52.239, -19.525, 97.93, 81.151, 53.139, -75.451]
  Call Extruder(410.87946)
  MoveL 8617 to (-41.29, 142.86, 125.68) mm, rotated rx 180 ry 0 rz 180 deg; joints [-52.09, -19.693, 98.044, 81.063, 53.003, -75.355]
  Call Extruder(452.94428)
  MoveL 8618 to (-41.29, 57.14, 125.68) mm, rotated rx 180 ry 0 rz 180 deg; joints [-40.759, -28.516, 103.344, 73.11, 43.024, -67.445]
  Call Extruder(453.37284)
  MoveL 8619 to (-41.27, 56.26, 125.68) mm, rotated rx 180 ry 0 rz 180 deg; joints [-40.614, -28.594, 103.385, 72.99, 42.902, -67.334]
  MoveL 8620 to (-41.27, 56.26, 125.68) mm, rotated rx 180 ry 0 rz 180 deg; joints [-40.614, -28.594, 103.385, 72.99, 42.902, -67.334]
  Call Extruder(453.94629)
  MoveL 8621 to (-41.22, 55.1, 125.68) mm, rotated rx 180 ry 0 rz 180 deg; joints [-40.419, -28.694, 103.437, 72.83, 42.735, -67.185]
  MoveL 8622 to (-41.22, 55.1, 125.68) mm, rotated rx 180 ry 0 rz 180 deg; joints [-40.419, -28.694, 103.437, 72.83, 42.735, -67.185]
  Call Extruder(454.38061)
  MoveL 8623 to (-41.18, 54.23, 125.68) mm, rotated rx 180 ry 0 rz 180 deg; joints [-40.269, -28.768, 103.476, 72.707, 42.608, -67.072]
  MoveL 8624 to (-41.18, 54.23, 125.68) mm, rotated rx 180 ry 0 rz 180 deg; joints [-40.269, -28.768, 103.476, 72.707, 42.608, -67.072]
  Call Extruder(454.67467)
  MoveL 8625 to (-41.13, 53.64, 125.68) mm, rotated rx -180 ry 0 rz 180 deg; joints [-40.165, -28.815, 103.501, 72.624, 42.519, -66.996]
  MoveL 8626 to (-41.13, 53.64, 125.68) mm, rotated rx -180 ry 0 rz 180 deg; joints [-40.165, -28.815, 103.501, 72.624, 42.519, -66.996]
  Call Extruder(454.97007)
  MoveL 8627 to (-41.09, 53.05, 125.68) mm, rotated rx 180 ry 0 rz 180 deg; joints [-40.062, -28.863, 103.526, 72.54, 42.431, -66.919]
  MoveL 8628 to (-41.09, 53.05, 125.68) mm, rotated rx 180 ry 0 rz 180 deg; joints [-40.062, -28.863, 103.526, 72.54, 42.431, -66.919]
  Call Extruder(455.21630)
  MoveL 8629 to (-41.04, 52.56, 125.68) mm, rotated rx 180 ry 0 rz 180 deg; joints [-39.975, -28.902, 103.546, 72.47, 42.356, -66.855]
  MoveL 8630 to (-41.04, 52.56, 125.68) mm, rotated rx 180 ry 0 rz 180 deg; joints [-39.975, -28.902, 103.546, 72.47, 42.356, -66.855]
  Call Extruder(455.41301)
  MoveL 8631 to (-40.99, 52.17, 125.68) mm, rotated rx 180 ry 0 rz -180 deg; joints [-39.904, -28.932, 103.561, 72.414, 42.296, -66.805]
  MoveL 8632 to (-40.99, 52.17, 125.68) mm, rotated rx 180 ry 0 rz -180 deg; joints [-39.904, -28.932, 103.561, 72.414, 42.296, -66.805]
  Call Extruder(455.61058)
  MoveL 8633 to (-40.95, 51.78, 125.68) mm, rotated rx 180 ry 0 rz 180 deg; joints [-39.833, -28.961, 103.577, 72.357, 42.235, -66.754]
  MoveL 8634 to (-40.95, 51.78, 125.68) mm, rotated rx 180 ry 0 rz 180 deg; joints [-39.833, -28.961, 103.577, 72.357, 42.235, -66.754]
  Call Extruder(455.80903)
  MoveL 8635 to (-40.9, 51.4, 125.68) mm, rotated rx -180 ry 0 rz 180 deg; joints [-39.763, -28.991, 103.592, 72.301, 42.174, -66.703]
  MoveL 8636 to (-40.9, 51.4, 125.68) mm, rotated rx -180 ry 0 rz 180 deg; joints [-39.763, -28.991, 103.592, 72.301, 42.174, -66.703]
  Call Extruder(456.00833)
  MoveL 8637 to (-40.86, 51.01, 125.68) mm, rotated rx 180 ry 0 rz 180 deg; joints [-39.692, -29.02, 103.607, 72.244, 42.114, -66.652]
  MoveL 8638 to (-40.86, 51.01, 125.68) mm, rotated rx 180 ry 0 rz 180 deg; joints [-39.692, -29.02, 103.607, 72.244, 42.114, -66.652]
  Call Extruder(456.16715)
  MoveL 8639 to (-40.81, 50.7, 125.68) mm, rotated rx 180 ry 0 rz 180 deg; joints [-39.634, -29.042, 103.618, 72.199, 42.064, -66.611]
  MoveL 8640 to (-40.81, 50.7, 125.68) mm, rotated rx 180 ry 0 rz 180 deg; joints [-39.634, -29.042, 103.618, 72.199, 42.064, -66.611]
  Call Extruder(456.32669)
  MoveL 8641 to (-40.76, 50.4, 125.68) mm, rotated rx 180 ry 0 rz 180 deg; joints [-39.576, -29.064, 103.63, 72.153, 42.014, -66.571]
  MoveL 8642 to (-40.76, 50.4, 125.68) mm, rotated rx 180 ry 0 rz 180 deg; joints [-39.576, -29.064, 103.63, 72.153, 42.014, -66.571]
  Call Extruder(456.48696)
  MoveL 8643 to (-40.71, 50.09, 125.68) mm, rotated rx 180 ry 0 rz 180 deg; joints [-39.518, -29.086, 103.641, 72.108, 41.964, -66.53]
  MoveL 8644 to (-40.71, 50.09, 125.68) mm, rotated rx 180 ry 0 rz 180 deg; joints [-39.518, -29.086, 103.641, 72.108, 41.964, -66.53]
  Call Extruder(456.64796)
  MoveL 8645 to (-40.66, 49.79, 125.68) mm, rotated rx 180 ry 0 rz 180 deg; joints [-39.46, -29.107, 103.652, 72.062, 41.914, -66.489]
  MoveL 8646 to (-40.66, 49.79, 125.68) mm, rotated rx 180 ry 0 rz 180 deg; joints [-39.46, -29.107, 103.652, 72.062, 41.914, -66.489]
  Call Extruder(456.80968)
  MoveL 8647 to (-40.61, 49.48, 125.68) mm, rotated rx 180 ry 0 rz 180 deg; joints [-39.402, -29.129, 103.663, 72.016, 41.864, -66.449]
  MoveL 8648 to (-40.61, 49.48, 125.68) mm, rotated rx 180 ry 0 rz 180 deg; joints [-39.402, -29.129, 103.663, 72.016, 41.864, -66.449]
  Call Extruder(456.97214)
  MoveL 8649 to (-40.56, 49.17, 125.68) mm, rotated rx 180 ry 0 rz 180 deg; joints [-39.344, -29.151, 103.675, 71.97, 41.814, -66.408]
  MoveL 8650 to (-40.56, 49.17, 125.68) mm, rotated rx 180 ry 0 rz 180 deg; joints [-39.344, -29.151, 103.675, 71.97, 41.814, -66.408]
  Call Extruder(457.10606)
  MoveL 8651 to (-40.52, 48.93, 125.68) mm, rotated rx 180 ry 0 rz 180 deg; joints [-39.296, -29.167, 103.683, 71.932, 41.772, -66.374]
  MoveL 8652 to (-40.52, 48.93, 125.68) mm, rotated rx 180 ry 0 rz 180 deg; joints [-39.296, -29.167, 103.683, 71.932, 41.772, -66.374]
  Call Extruder(457.24060)
  MoveL 8653 to (-40.47, 48.68, 125.68) mm, rotated rx -180 ry 0 rz 180 deg; joints [-39.247, -29.184, 103.692, 71.894, 41.73, -66.341]
  MoveL 8654 to (-40.47, 48.68, 125.68) mm, rotated rx -180 ry 0 rz 180 deg; joints [-39.247, -29.184, 103.692, 71.894, 41.73, -66.341]
  Call Extruder(457.37574)
  MoveL 8655 to (-40.42, 48.43, 125.68) mm, rotated rx 180 ry 0 rz 180 deg; joints [-39.198, -29.2, 103.7, 71.856, 41.688, -66.307]
  MoveL 8656 to (-40.42, 48.43, 125.68) mm, rotated rx 180 ry 0 rz 180 deg; joints [-39.198, -29.2, 103.7, 71.856, 41.688, -66.307]
  Call Extruder(457.51150)
  MoveL 8657 to (-40.37, 48.18, 125.68) mm, rotated rx 180 ry 0 rz 180 deg; joints [-39.149, -29.217, 103.709, 71.818, 41.646, -66.274]
  MoveL 8658 to (-40.37, 48.18, 125.68) mm, rotated rx 180 ry 0 rz 180 deg; joints [-39.149, -29.217, 103.709, 71.818, 41.646, -66.274]
  Call Extruder(457.64786)
  MoveL 8659 to (-40.32, 47.93, 125.68) mm, rotated rx 180 ry 0 rz 180 deg; joints [-39.1, -29.233, 103.717, 71.78, 41.603, -66.24]
  MoveL 8660 to (-40.32, 47.93, 125.68) mm, rotated rx 180 ry 0 rz 180 deg; joints [-39.1, -29.233, 103.717, 71.78, 41.603, -66.24]
  Call Extruder(457.78484)
  MoveL 8661 to (-40.27, 47.68, 125.68) mm, rotated rx -180 ry 0 rz -180 deg; joints [-39.051, -29.25, 103.725, 71.742, 41.561, -66.207]
  MoveL 8662 to (-40.27, 47.68, 125.68) mm, rotated rx -180 ry 0 rz -180 deg; joints [-39.051, -29.25, 103.725, 71.742, 41.561, -66.207]
  Call Extruder(457.92243)
  MoveL 8663 to (-40.22, 47.43, 125.68) mm, rotated rx 180 ry 0 rz -180 deg; joints [-39.002, -29.266, 103.734, 71.703, 41.519, -66.173]
  MoveL 8664 to (-40.22, 47.43, 125.68) mm, rotated rx 180 ry 0 rz -180 deg; joints [-39.002, -29.266, 103.734, 71.703, 41.519, -66.173]
  Call Extruder(458.03615)
  MoveL 8665 to (-40.17, 47.23, 125.68) mm, rotated rx 180 ry 0 rz 180 deg; joints [-38.962, -29.279, 103.74, 71.672, 41.483, -66.145]
  MoveL 8666 to (-40.17, 47.23, 125.68) mm, rotated rx 180 ry 0 rz 180 deg; joints [-38.962, -29.279, 103.74, 71.672, 41.483, -66.145]
  Call Extruder(458.15034)
  MoveL 8667 to (-40.13, 47.02, 125.68) mm, rotated rx 180 ry 0 rz 180 deg; joints [-38.921, -29.292, 103.747, 71.64, 41.448, -66.117]
  MoveL 8668 to (-40.13, 47.02, 125.68) mm, rotated rx 180 ry 0 rz 180 deg; joints [-38.921, -29.292, 103.747, 71.64, 41.448, -66.117]
  Call Extruder(458.26497)
  MoveL 8669 to (-40.08, 46.82, 125.68) mm, rotated rx -180 ry 0 rz 180 deg; joints [-38.88, -29.305, 103.754, 71.608, 41.413, -66.09]
  MoveL 8670 to (-40.08, 46.82, 125.68) mm, rotated rx -180 ry 0 rz 180 deg; joints [-38.88, -29.305, 103.754, 71.608, 41.413, -66.09]
  Call Extruder(458.38006)
  MoveL 8671 to (-40.04, 46.61, 125.68) mm, rotated rx 180 ry 0 rz 180 deg; joints [-38.839, -29.318, 103.76, 71.576, 41.377, -66.062]
  MoveL 8672 to (-40.04, 46.61, 125.68) mm, rotated rx 180 ry 0 rz 180 deg; joints [-38.839, -29.318, 103.76, 71.576, 41.377, -66.062]
  Call Extruder(458.50230)
  MoveL 8673 to (-39.98, 46.4, 125.68) mm, rotated rx -180 ry 0 rz -180 deg; joints [-38.795, -29.331, 103.767, 71.542, 41.339, -66.033]
  MoveL 8674 to (-39.98, 46.4, 125.68) mm, rotated rx -180 ry 0 rz -180 deg; joints [-38.795, -29.331, 103.767, 71.542, 41.339, -66.033]
  Call Extruder(458.63196)
  MoveL 8675 to (-39.92, 46.18, 125.68) mm, rotated rx 180 ry 0 rz 180 deg; joints [-38.748, -29.343, 103.773, 71.507, 41.298, -66.002]
  MoveL 8676 to (-39.92, 46.18, 125.68) mm, rotated rx 180 ry 0 rz 180 deg; joints [-38.748, -29.343, 103.773, 71.507, 41.298, -66.002]
  Call Extruder(458.76219)
  MoveL 8677 to (-39.85, 45.95, 125.68) mm, rotated rx 180 ry 0 rz 180 deg; joints [-38.7, -29.355, 103.779, 71.471, 41.256, -65.972]
  MoveL 8678 to (-39.85, 45.95, 125.68) mm, rotated rx 180 ry 0 rz 180 deg; joints [-38.7, -29.355, 103.779, 71.471, 41.256, -65.972]
  Call Extruder(458.89299)
  MoveL 8679 to (-39.78, 45.73, 125.68) mm, rotated rx 180 ry 0 rz 180 deg; joints [-38.653, -29.367, 103.785, 71.436, 41.215, -65.941]
  MoveL 8680 to (-39.78, 45.73, 125.68) mm, rotated rx 180 ry 0 rz 180 deg; joints [-38.653, -29.367, 103.785, 71.436, 41.215, -65.941]
  Call Extruder(459.02435)
  MoveL 8681 to (-39.71, 45.51, 125.68) mm, rotated rx -180 ry 0 rz 180 deg; joints [-38.605, -29.379, 103.791, 71.4, 41.173, -65.911]
  MoveL 8682 to (-39.71, 45.51, 125.68) mm, rotated rx -180 ry 0 rz 180 deg; joints [-38.605, -29.379, 103.791, 71.4, 41.173, -65.911]
  Call Extruder(459.13625)
  MoveL 8683 to (-39.65, 45.32, 125.68) mm, rotated rx 180 ry 0 rz -180 deg; joints [-38.565, -29.388, 103.796, 71.37, 41.138, -65.885]
  MoveL 8684 to (-39.65, 45.32, 125.68) mm, rotated rx 180 ry 0 rz -180 deg; joints [-38.565, -29.388, 103.796, 71.37, 41.138, -65.885]
  Call Extruder(459.24859)
  MoveL 8685 to (-39.59, 45.13, 125.68) mm, rotated rx 180 ry 0 rz 180 deg; joints [-38.524, -29.398, 103.801, 71.339, 41.102, -65.859]
  MoveL 8686 to (-39.59, 45.13, 125.68) mm, rotated rx 180 ry 0 rz 180 deg; joints [-38.524, -29.398, 103.801, 71.339, 41.102, -65.859]
  Call Extruder(459.36138)
  MoveL 8687 to (-39.53, 44.94, 125.68) mm, rotated rx -180 ry 0 rz 180 deg; joints [-38.483, -29.408, 103.806, 71.309, 41.067, -65.833]
  MoveL 8688 to (-39.53, 44.94, 125.68) mm, rotated rx -180 ry 0 rz 180 deg; joints [-38.483, -29.408, 103.806, 71.309, 41.067, -65.833]
  Call Extruder(459.47461)
  MoveL 8689 to (-39.47, 44.75, 125.68) mm, rotated rx -180 ry 0 rz 180 deg; joints [-38.443, -29.417, 103.811, 71.278, 41.031, -65.807]
  MoveL 8690 to (-39.47, 44.75, 125.68) mm, rotated rx -180 ry 0 rz 180 deg; joints [-38.443, -29.417, 103.811, 71.278, 41.031, -65.807]
  Call Extruder(459.58829)
  MoveL 8691 to (-39.41, 44.56, 125.68) mm, rotated rx 180 ry 0 rz 180 deg; joints [-38.402, -29.427, 103.816, 71.248, 40.995, -65.781]
  MoveL 8692 to (-39.41, 44.56, 125.68) mm, rotated rx 180 ry 0 rz 180 deg; joints [-38.402, -29.427, 103.816, 71.248, 40.995, -65.781]
  Call Extruder(459.77026)
  MoveL 8693 to (-39.29, 44.27, 125.68) mm, rotated rx 180 ry 0 rz 180 deg; joints [-38.335, -29.439, 103.822, 71.2, 40.937, -65.741]
  MoveL 8694 to (-39.29, 44.27, 125.68) mm, rotated rx 180 ry 0 rz 180 deg; joints [-38.335, -29.439, 103.822, 71.2, 40.937, -65.741]
  Call Extruder(459.95298)
  MoveL 8695 to (-39.17, 43.98, 125.68) mm, rotated rx 180 ry 0 rz 180 deg; joints [-38.269, -29.451, 103.828, 71.151, 40.878, -65.701]
  MoveL 8696 to (-39.17, 43.98, 125.68) mm, rotated rx 180 ry 0 rz 180 deg; joints [-38.269, -29.451, 103.828, 71.151, 40.878, -65.701]
  Call Extruder(460.12339)
  MoveL 8697 to (-39.05, 43.71, 125.68) mm, rotated rx 180 ry 0 rz 180 deg; joints [-38.207, -29.461, 103.834, 71.107, 40.823, -65.664]
  MoveL 8698 to (-39.05, 43.71, 125.68) mm, rotated rx 180 ry 0 rz 180 deg; joints [-38.207, -29.461, 103.834, 71.107, 40.823, -65.664]
  Call Extruder(460.28137)
  MoveL 8699 to (-38.94, 43.46, 125.68) mm, rotated rx 180 ry 0 rz 180 deg; joints [-38.149, -29.471, 103.838, 71.065, 40.772, -65.63]
  MoveL 8700 to (-38.94, 43.46, 125.68) mm, rotated rx 180 ry 0 rz 180 deg; joints [-38.149, -29.471, 103.838, 71.065, 40.772, -65.63]
  Call Extruder(460.43996)
  MoveL 8701 to (-38.84, 43.21, 125.68) mm, rotated rx -180 ry 0 rz 180 deg; joints [-38.092, -29.481, 103.843, 71.023, 40.721, -65.595]
  MoveL 8702 to (-38.84, 43.21, 125.68) mm, rotated rx -180 ry 0 rz 180 deg; joints [-38.092, -29.481, 103.843, 71.023, 40.721, -65.595]
  Call Extruder(460.64612)
  MoveL 8703 to (-38.66, 42.91, 125.68) mm, rotated rx -180 ry 0 rz 180 deg; joints [-38.016, -29.488, 103.847, 70.971, 40.653, -65.554]
  MoveL 8704 to (-38.66, 42.91, 125.68) mm, rotated rx -180 ry 0 rz 180 deg; joints [-38.016, -29.488, 103.847, 70.971, 40.653, -65.554]
  Call Extruder(460.85306)
  MoveL 8705 to (-38.49, 42.6, 125.68) mm, rotated rx -180 ry 0 rz 180 deg; joints [-37.939, -29.494, 103.85, 70.919, 40.584, -65.512]
  MoveL 8706 to (-38.49, 42.6, 125.68) mm, rotated rx -180 ry 0 rz 180 deg; joints [-37.939, -29.494, 103.85, 70.919, 40.584, -65.512]
  Call Extruder(461.06079)
  MoveL 8707 to (-38.31, 42.3, 125.68) mm, rotated rx 180 ry 0 rz -180 deg; joints [-37.863, -29.501, 103.854, 70.867, 40.516, -65.47]
  MoveL 8708 to (-38.31, 42.3, 125.68) mm, rotated rx 180 ry 0 rz -180 deg; joints [-37.863, -29.501, 103.854, 70.867, 40.516, -65.47]
  Call Extruder(461.26929)
  MoveL 8709 to (-38.14, 41.99, 125.68) mm, rotated rx 180 ry 0 rz 180 deg; joints [-37.787, -29.508, 103.857, 70.814, 40.448, -65.428]
  MoveL 8710 to (-38.14, 41.99, 125.68) mm, rotated rx 180 ry 0 rz 180 deg; joints [-37.787, -29.508, 103.857, 70.814, 40.448, -65.428]
  Call Extruder(461.44884)
  MoveL 8711 to (-37.96, 41.75, 125.68) mm, rotated rx -180 ry 0 rz -180 deg; joints [-37.72, -29.509, 103.858, 70.771, 40.388, -65.395]
  MoveL 8712 to (-37.96, 41.75, 125.68) mm, rotated rx -180 ry 0 rz -180 deg; joints [-37.72, -29.509, 103.858, 70.771, 40.388, -65.395]
  Call Extruder(461.78228)
  MoveL 8713 to (-37.63, 41.3, 125.68) mm, rotated rx 180 ry 0 rz 180 deg; joints [-37.598, -29.511, 103.859, 70.691, 40.277, -65.333]
  MoveL 8714 to (-37.63, 41.3, 125.68) mm, rotated rx 180 ry 0 rz 180 deg; joints [-37.598, -29.511, 103.859, 70.691, 40.277, -65.333]
  Call Extruder(462.11690)
  MoveL 8715 to (-37.3, 40.85, 125.68) mm, rotated rx 180 ry 0 rz 180 deg; joints [-37.475, -29.514, 103.86, 70.611, 40.166, -65.271]
  Call Extruder(462.94483)
  MoveL 8716 to (-36.39, 39.81, 125.68) mm, rotated rx 180 ry 0 rz 180 deg; joints [-37.173, -29.5, 103.853, 70.421, 39.889, -65.13]
  Call Extruder(463.77274)
  MoveL 8717 to (-35.35, 38.9, 125.68) mm, rotated rx 180 ry 0 rz 180 deg; joints [-36.876, -29.462, 103.834, 70.246, 39.614, -65.007]
  Call Extruder(463.94004)
  MoveL 8718 to (-35.13, 38.73, 125.68) mm, rotated rx 180 ry 0 rz 180 deg; joints [-36.818, -29.45, 103.828, 70.214, 39.559, -64.986]
  MoveL 8719 to (-35.13, 38.73, 125.68) mm, rotated rx 180 ry 0 rz 180 deg; joints [-36.818, -29.45, 103.828, 70.214, 39.559, -64.986]
  Call Extruder(464.27347)
  MoveL 8720 to (-34.68, 38.41, 125.68) mm, rotated rx 180 ry 0 rz 180 deg; joints [-36.701, -29.427, 103.816, 70.149, 39.449, -64.942]
  MoveL 8721 to (-34.68, 38.41, 125.68) mm, rotated rx 180 ry 0 rz 180 deg; joints [-36.701, -29.427, 103.816, 70.149, 39.449, -64.942]
  Call Extruder(464.60571)
  MoveL 8722 to (-34.22, 38.08, 125.68) mm, rotated rx 180 ry 0 rz 180 deg; joints [-36.584, -29.404, 103.804, 70.084, 39.339, -64.899]
  MoveL 8723 to (-34.22, 38.08, 125.68) mm, rotated rx 180 ry 0 rz 180 deg; joints [-36.584, -29.404, 103.804, 70.084, 39.339, -64.899]
  Call Extruder(464.72342)
  MoveL 8724 to (-34.05, 37.98, 125.68) mm, rotated rx 180 ry 0 rz 180 deg; joints [-36.544, -29.393, 103.799, 70.064, 39.302, -64.886]
  MoveL 8725 to (-34.05, 37.98, 125.68) mm, rotated rx 180 ry 0 rz 180 deg; joints [-36.544, -29.393, 103.799, 70.064, 39.302, -64.886]
  Call Extruder(464.93114)
  MoveL 8726 to (-33.75, 37.8, 125.68) mm, rotated rx 180 ry 0 rz 180 deg; joints [-36.474, -29.374, 103.789, 70.027, 39.234, -64.863]
  MoveL 8727 to (-33.75, 37.8, 125.68) mm, rotated rx 180 ry 0 rz 180 deg; joints [-36.474, -29.374, 103.789, 70.027, 39.234, -64.863]
  Call Extruder(465.13808)
  MoveL 8728 to (-33.45, 37.63, 125.68) mm, rotated rx 180 ry 0 rz 180 deg; joints [-36.403, -29.355, 103.779, 69.991, 39.168, -64.841]
  MoveL 8729 to (-33.45, 37.63, 125.68) mm, rotated rx 180 ry 0 rz 180 deg; joints [-36.403, -29.355, 103.779, 69.991, 39.168, -64.841]
  Call Extruder(465.34424)
  MoveL 8730 to (-33.14, 37.45, 125.68) mm, rotated rx 180 ry 0 rz 180 deg; joints [-36.333, -29.335, 103.769, 69.955, 39.101, -64.819]
  MoveL 8731 to (-33.14, 37.45, 125.68) mm, rotated rx 180 ry 0 rz 180 deg; joints [-36.333, -29.335, 103.769, 69.955, 39.101, -64.819]
  Call Extruder(465.52591)
  MoveL 8732 to (-32.86, 37.31, 125.68) mm, rotated rx 180 ry 0 rz -180 deg; joints [-36.272, -29.316, 103.759, 69.924, 39.042, -64.801]
  MoveL 8733 to (-32.86, 37.31, 125.68) mm, rotated rx 180 ry 0 rz -180 deg; joints [-36.272, -29.316, 103.759, 69.924, 39.042, -64.801]
  Call Extruder(465.68390)
  MoveL 8734 to (-32.62, 37.2, 125.68) mm, rotated rx -180 ry 0 rz 180 deg; joints [-36.221, -29.297, 103.749, 69.901, 38.993, -64.788]
  MoveL 8735 to (-32.62, 37.2, 125.68) mm, rotated rx -180 ry 0 rz 180 deg; joints [-36.221, -29.297, 103.749, 69.901, 38.993, -64.788]
  Call Extruder(465.84129)
  MoveL 8736 to (-32.37, 37.1, 125.68) mm, rotated rx -180 ry 0 rz 180 deg; joints [-36.17, -29.278, 103.74, 69.877, 38.944, -64.775]
  MoveL 8737 to (-32.37, 37.1, 125.68) mm, rotated rx -180 ry 0 rz 180 deg; joints [-36.17, -29.278, 103.74, 69.877, 38.944, -64.775]
  Call Extruder(465.98171)
  MoveL 8738 to (-32.14, 37, 125.68) mm, rotated rx 180 ry 0 rz 180 deg; joints [-36.125, -29.26, 103.731, 69.856, 38.9, -64.764]
  MoveL 8739 to (-32.14, 37, 125.68) mm, rotated rx 180 ry 0 rz 180 deg; joints [-36.125, -29.26, 103.731, 69.856, 38.9, -64.764]
  Call Extruder(466.13359)
  MoveL 8740 to (-31.9, 36.9, 125.68) mm, rotated rx 180 ry 0 rz 180 deg; joints [-36.076, -29.241, 103.721, 69.834, 38.853, -64.752]
  MoveL 8741 to (-31.9, 36.9, 125.68) mm, rotated rx 180 ry 0 rz 180 deg; joints [-36.076, -29.241, 103.721, 69.834, 38.853, -64.752]
  Call Extruder(466.29670)
  MoveL 8742 to (-31.64, 36.79, 125.68) mm, rotated rx 180 ry 0 rz 180 deg; joints [-36.023, -29.221, 103.71, 69.809, 38.801, -64.739]
  MoveL 8743 to (-31.64, 36.79, 125.68) mm, rotated rx 180 ry 0 rz 180 deg; joints [-36.023, -29.221, 103.71, 69.809, 38.801, -64.739]
  Call Extruder(466.41015)
  MoveL 8744 to (-31.45, 36.73, 125.68) mm, rotated rx 180 ry 0 rz 180 deg; joints [-35.989, -29.204, 103.702, 69.795, 38.767, -64.732]
  MoveL 8745 to (-31.45, 36.73, 125.68) mm, rotated rx 180 ry 0 rz 180 deg; joints [-35.989, -29.204, 103.702, 69.795, 38.767, -64.732]
  Call Extruder(466.52317)
  MoveL 8746 to (-31.26, 36.67, 125.68) mm, rotated rx 180 ry 0 rz 180 deg; joints [-35.954, -29.188, 103.694, 69.78, 38.733, -64.725]
  MoveL 8747 to (-31.26, 36.67, 125.68) mm, rotated rx 180 ry 0 rz 180 deg; joints [-35.954, -29.188, 103.694, 69.78, 38.733, -64.725]
  Call Extruder(466.63573)
  MoveL 8748 to (-31.07, 36.61, 125.68) mm, rotated rx 180 ry 0 rz 180 deg; joints [-35.919, -29.172, 103.686, 69.766, 38.699, -64.718]
  MoveL 8749 to (-31.07, 36.61, 125.68) mm, rotated rx 180 ry 0 rz 180 deg; joints [-35.919, -29.172, 103.686, 69.766, 38.699, -64.718]
  Call Extruder(466.74786)
  MoveL 8750 to (-30.88, 36.55, 125.68) mm, rotated rx 180 ry 0 rz 180 deg; joints [-35.884, -29.156, 103.677, 69.751, 38.664, -64.711]
  MoveL 8751 to (-30.88, 36.55, 125.68) mm, rotated rx 180 ry 0 rz 180 deg; joints [-35.884, -29.156, 103.677, 69.751, 38.664, -64.711]
  Call Extruder(466.85954)
  MoveL 8752 to (-30.69, 36.49, 125.68) mm, rotated rx 180 ry 0 rz 180 deg; joints [-35.849, -29.14, 103.669, 69.736, 38.63, -64.705]
  MoveL 8753 to (-30.69, 36.49, 125.68) mm, rotated rx 180 ry 0 rz 180 deg; joints [-35.849, -29.14, 103.669, 69.736, 38.63, -64.705]
  Call Extruder(466.99061)
  MoveL 8754 to (-30.47, 36.42, 125.68) mm, rotated rx -180 ry 0 rz 180 deg; joints [-35.809, -29.12, 103.659, 69.72, 38.59, -64.697]
  MoveL 8755 to (-30.47, 36.42, 125.68) mm, rotated rx -180 ry 0 rz 180 deg; joints [-35.809, -29.12, 103.659, 69.72, 38.59, -64.697]
  Call Extruder(467.12112)
  MoveL 8756 to (-30.25, 36.35, 125.68) mm, rotated rx 180 ry 0 rz 180 deg; joints [-35.768, -29.1, 103.649, 69.704, 38.551, -64.69]
  MoveL 8757 to (-30.25, 36.35, 125.68) mm, rotated rx 180 ry 0 rz 180 deg; joints [-35.768, -29.1, 103.649, 69.704, 38.551, -64.69]
  Call Extruder(467.25107)
  MoveL 8758 to (-30.02, 36.28, 125.68) mm, rotated rx 180 ry 0 rz -180 deg; joints [-35.728, -29.081, 103.638, 69.687, 38.511, -64.683]
  MoveL 8759 to (-30.02, 36.28, 125.68) mm, rotated rx 180 ry 0 rz -180 deg; joints [-35.728, -29.081, 103.638, 69.687, 38.511, -64.683]
  Call Extruder(467.38045)
  MoveL 8760 to (-29.8, 36.22, 125.68) mm, rotated rx 180 ry 0 rz 180 deg; joints [-35.688, -29.061, 103.628, 69.671, 38.471, -64.676]
  MoveL 8761 to (-29.8, 36.22, 125.68) mm, rotated rx 180 ry 0 rz 180 deg; joints [-35.688, -29.061, 103.628, 69.671, 38.471, -64.676]
  Call Extruder(467.50241)
  MoveL 8762 to (-29.59, 36.16, 125.68) mm, rotated rx -180 ry 0 rz 180 deg; joints [-35.651, -29.041, 103.618, 69.656, 38.434, -64.67]
  MoveL 8763 to (-29.59, 36.16, 125.68) mm, rotated rx -180 ry 0 rz 180 deg; joints [-35.651, -29.041, 103.618, 69.656, 38.434, -64.67]
  Call Extruder(467.61726)
  MoveL 8764 to (-29.38, 36.12, 125.68) mm, rotated rx 180 ry 0 rz 180 deg; joints [-35.617, -29.022, 103.608, 69.644, 38.401, -64.666]
  MoveL 8765 to (-29.38, 36.12, 125.68) mm, rotated rx 180 ry 0 rz 180 deg; joints [-35.617, -29.022, 103.608, 69.644, 38.401, -64.666]
  Call Extruder(467.73165)
  MoveL 8766 to (-29.18, 36.07, 125.68) mm, rotated rx -180 ry 0 rz 180 deg; joints [-35.584, -29.003, 103.598, 69.632, 38.367, -64.662]
  MoveL 8767 to (-29.18, 36.07, 125.68) mm, rotated rx -180 ry 0 rz 180 deg; joints [-35.584, -29.003, 103.598, 69.632, 38.367, -64.662]
  Call Extruder(467.84560)
  MoveL 8768 to (-28.97, 36.03, 125.68) mm, rotated rx -180 ry 0 rz 180 deg; joints [-35.55, -28.983, 103.588, 69.62, 38.334, -64.658]
  MoveL 8769 to (-28.97, 36.03, 125.68) mm, rotated rx -180 ry 0 rz 180 deg; joints [-35.55, -28.983, 103.588, 69.62, 38.334, -64.658]
  Call Extruder(467.95909)
  MoveL 8770 to (-28.77, 35.98, 125.68) mm, rotated rx 180 ry 0 rz 180 deg; joints [-35.517, -28.964, 103.578, 69.608, 38.3, -64.654]
  MoveL 8771 to (-28.77, 35.98, 125.68) mm, rotated rx 180 ry 0 rz 180 deg; joints [-35.517, -28.964, 103.578, 69.608, 38.3, -64.654]
  Call Extruder(468.09637)
  MoveL 8772 to (-28.52, 35.93, 125.68) mm, rotated rx 180 ry 0 rz 180 deg; joints [-35.477, -28.94, 103.565, 69.594, 38.26, -64.65]
  MoveL 8773 to (-28.52, 35.93, 125.68) mm, rotated rx 180 ry 0 rz 180 deg; joints [-35.477, -28.94, 103.565, 69.594, 38.26, -64.65]
  Call Extruder(468.23304)
  MoveL 8774 to (-28.27, 35.88, 125.68) mm, rotated rx 180 ry 0 rz 180 deg; joints [-35.437, -28.915, 103.553, 69.581, 38.22, -64.646]
  MoveL 8775 to (-28.27, 35.88, 125.68) mm, rotated rx 180 ry 0 rz 180 deg; joints [-35.437, -28.915, 103.553, 69.581, 38.22, -64.646]
  Call Extruder(468.36910)
  MoveL 8776 to (-28.02, 35.83, 125.68) mm, rotated rx 180 ry 0 rz 180 deg; joints [-35.397, -28.891, 103.54, 69.567, 38.18, -64.642]
  MoveL 8777 to (-28.02, 35.83, 125.68) mm, rotated rx 180 ry 0 rz 180 deg; joints [-35.397, -28.891, 103.54, 69.567, 38.18, -64.642]
  Call Extruder(468.50456)
  MoveL 8778 to (-27.77, 35.78, 125.68) mm, rotated rx -180 ry 0 rz 180 deg; joints [-35.357, -28.867, 103.528, 69.553, 38.14, -64.638]
  MoveL 8779 to (-27.77, 35.78, 125.68) mm, rotated rx -180 ry 0 rz 180 deg; joints [-35.357, -28.867, 103.528, 69.553, 38.14, -64.638]
  Call Extruder(468.63940)
  MoveL 8780 to (-27.52, 35.73, 125.68) mm, rotated rx 180 ry 0 rz 180 deg; joints [-35.317, -28.843, 103.515, 69.539, 38.099, -64.634]
  MoveL 8781 to (-27.52, 35.73, 125.68) mm, rotated rx 180 ry 0 rz 180 deg; joints [-35.317, -28.843, 103.515, 69.539, 38.099, -64.634]
  Call Extruder(468.77363)
  MoveL 8782 to (-27.27, 35.68, 125.68) mm, rotated rx 180 ry 0 rz 180 deg; joints [-35.277, -28.819, 103.503, 69.526, 38.059, -64.63]
  MoveL 8783 to (-27.27, 35.68, 125.68) mm, rotated rx 180 ry 0 rz 180 deg; joints [-35.277, -28.819, 103.503, 69.526, 38.059, -64.63]
  Call Extruder(468.90725)
  MoveL 8784 to (-27.03, 35.64, 125.68) mm, rotated rx 180 ry 0 rz 180 deg; joints [-35.238, -28.794, 103.49, 69.512, 38.02, -64.626]
  MoveL 8785 to (-27.03, 35.64, 125.68) mm, rotated rx 180 ry 0 rz 180 deg; joints [-35.238, -28.794, 103.49, 69.512, 38.02, -64.626]
  Call Extruder(469.06935)
  MoveL 8786 to (-26.72, 35.59, 125.68) mm, rotated rx 180 ry 0 rz 180 deg; joints [-35.191, -28.764, 103.474, 69.497, 37.972, -64.622]
  MoveL 8787 to (-26.72, 35.59, 125.68) mm, rotated rx 180 ry 0 rz 180 deg; joints [-35.191, -28.764, 103.474, 69.497, 37.972, -64.622]
  Call Extruder(469.23072)
  MoveL 8788 to (-26.41, 35.54, 125.68) mm, rotated rx 180 ry 0 rz 180 deg; joints [-35.145, -28.733, 103.458, 69.483, 37.925, -64.619]
  MoveL 8789 to (-26.41, 35.54, 125.68) mm, rotated rx 180 ry 0 rz 180 deg; joints [-35.145, -28.733, 103.458, 69.483, 37.925, -64.619]
  Call Extruder(469.39136)
  MoveL 8790 to (-26.11, 35.49, 125.68) mm, rotated rx 180 ry 0 rz -180 deg; joints [-35.098, -28.702, 103.442, 69.468, 37.878, -64.616]
  MoveL 8791 to (-26.11, 35.49, 125.68) mm, rotated rx 180 ry 0 rz -180 deg; joints [-35.098, -28.702, 103.442, 69.468, 37.878, -64.616]
  Call Extruder(469.55127)
  MoveL 8792 to (-25.8, 35.44, 125.68) mm, rotated rx 180 ry 0 rz 180 deg; joints [-35.052, -28.671, 103.426, 69.454, 37.831, -64.613]
  MoveL 8793 to (-25.8, 35.44, 125.68) mm, rotated rx 180 ry 0 rz 180 deg; joints [-35.052, -28.671, 103.426, 69.454, 37.831, -64.613]
  Call Extruder(469.71046)
  MoveL 8794 to (-25.5, 35.39, 125.68) mm, rotated rx -180 ry 0 rz 180 deg; joints [-35.006, -28.64, 103.409, 69.439, 37.784, -64.61]
  MoveL 8795 to (-25.5, 35.39, 125.68) mm, rotated rx -180 ry 0 rz 180 deg; joints [-35.006, -28.64, 103.409, 69.439, 37.784, -64.61]
  Call Extruder(469.86892)
  MoveL 8796 to (-25.19, 35.34, 125.68) mm, rotated rx 180 ry 0 rz -180 deg; joints [-34.96, -28.609, 103.393, 69.425, 37.738, -64.607]
  MoveL 8797 to (-25.19, 35.34, 125.68) mm, rotated rx 180 ry 0 rz -180 deg; joints [-34.96, -28.609, 103.393, 69.425, 37.738, -64.607]
  Call Extruder(470.06779)
  MoveL 8798 to (-24.8, 35.3, 125.68) mm, rotated rx -180 ry 0 rz 180 deg; joints [-34.904, -28.569, 103.372, 69.409, 37.681, -64.606]
  MoveL 8799 to (-24.8, 35.3, 125.68) mm, rotated rx -180 ry 0 rz 180 deg; joints [-34.904, -28.569, 103.372, 69.409, 37.681, -64.606]
  Call Extruder(470.26580)
  MoveL 8800 to (-24.42, 35.25, 125.68) mm, rotated rx 180 ry 0 rz 180 deg; joints [-34.849, -28.528, 103.351, 69.393, 37.624, -64.605]
  MoveL 8801 to (-24.42, 35.25, 125.68) mm, rotated rx 180 ry 0 rz 180 deg; joints [-34.849, -28.528, 103.351, 69.393, 37.624, -64.605]
  Call Extruder(470.46294)
